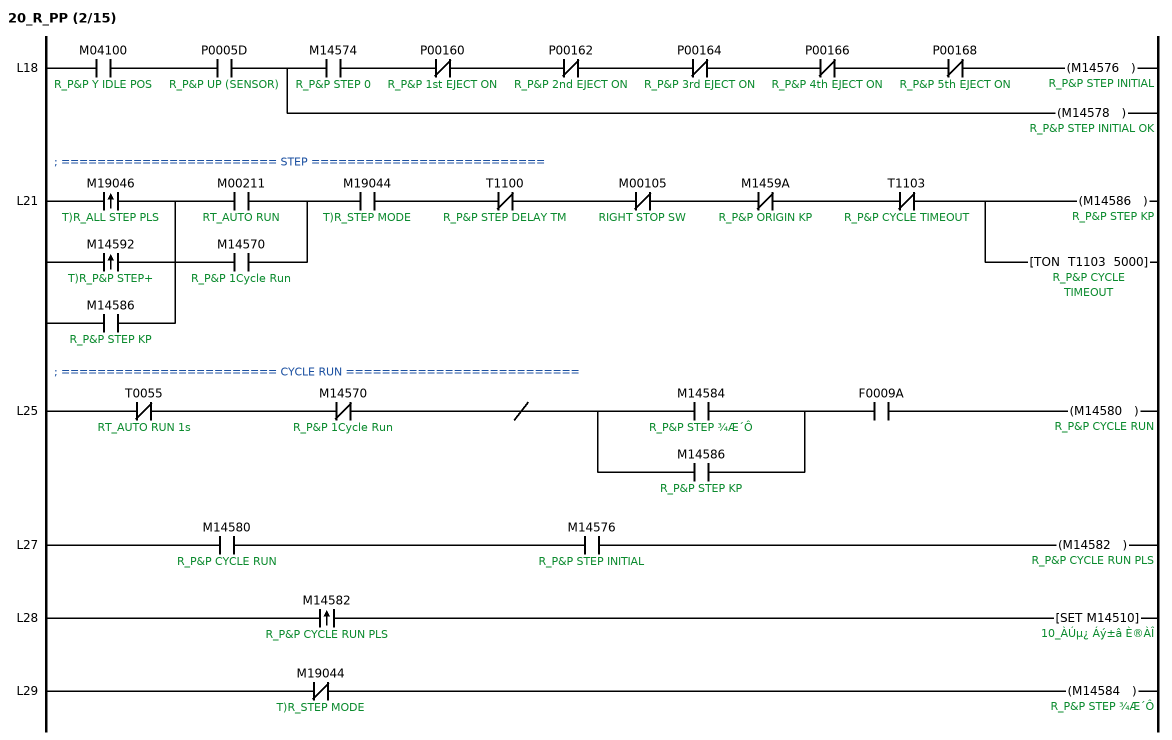
[picture p192: 20_R_PP rungs L18-L29]
; L18
LOAD      M04100	// R_P&P Y IDLE POS
AND       P0005D	// R_P&P UP (SENSOR)
MPUSH
AND       M14574	// R_P&P STEP 0
AND NOT   P00160	// R_P&P 1st EJECT ON
AND NOT   P00162	// R_P&P 2nd EJECT ON
AND NOT   P00164	// R_P&P 3rd EJECT ON
AND NOT   P00166	// R_P&P 4th EJECT ON
AND NOT   P00168	// R_P&P 5th EJECT ON
OUT       M14576	// R_P&P STEP INITIAL
MPOP
OUT       M14578	// R_P&P STEP INITIAL OK
// ======================== STEP ==========================
; L21
LOADP     M19046	// T)R_ALL STEP PLS
ORP       M14592	// T)R_P&P STEP+
OR        M14586	// R_P&P STEP KP
LOAD      M00211	// RT_AUTO RUN
OR        M14570	// R_P&P 1Cycle Run
AND LOAD
AND       M19044	// T)R_STEP MODE
AND NOT   T1100	// R_P&P STEP DELAY TM
AND NOT   M00105	// RIGHT STOP SW
AND NOT   M1459A	// R_P&P ORIGIN KP
AND NOT   T1103	// R_P&P CYCLE TIMEOUT
OUT       M14586	// R_P&P STEP KP
TON       T1103 5000	// R_P&P CYCLE TIMEOUT
// ======================== CYCLE RUN ==========================
; L25
LOAD NOT  T0055	// RT_AUTO RUN 1s
AND NOT   M14570	// R_P&P 1Cycle Run
NOT
LOAD      M14584	// R_P&P STEP ¾Æ´Ô
OR        M14586	// R_P&P STEP KP
AND LOAD
AND       F0009A
OUT       M14580	// R_P&P CYCLE RUN
; L27
LOAD      M14580	// R_P&P CYCLE RUN
AND       M14576	// R_P&P STEP INITIAL
OUT       M14582	// R_P&P CYCLE RUN PLS
; L28
LOADP     M14582	// R_P&P CYCLE RUN PLS
SET       M14510	// 10_ÀÚµ¿ Áý±â È®ÀÎ
; L29
LOAD NOT  M19044	// T)R_STEP MODE
OUT       M14584	// R_P&P STEP ¾Æ´Ô

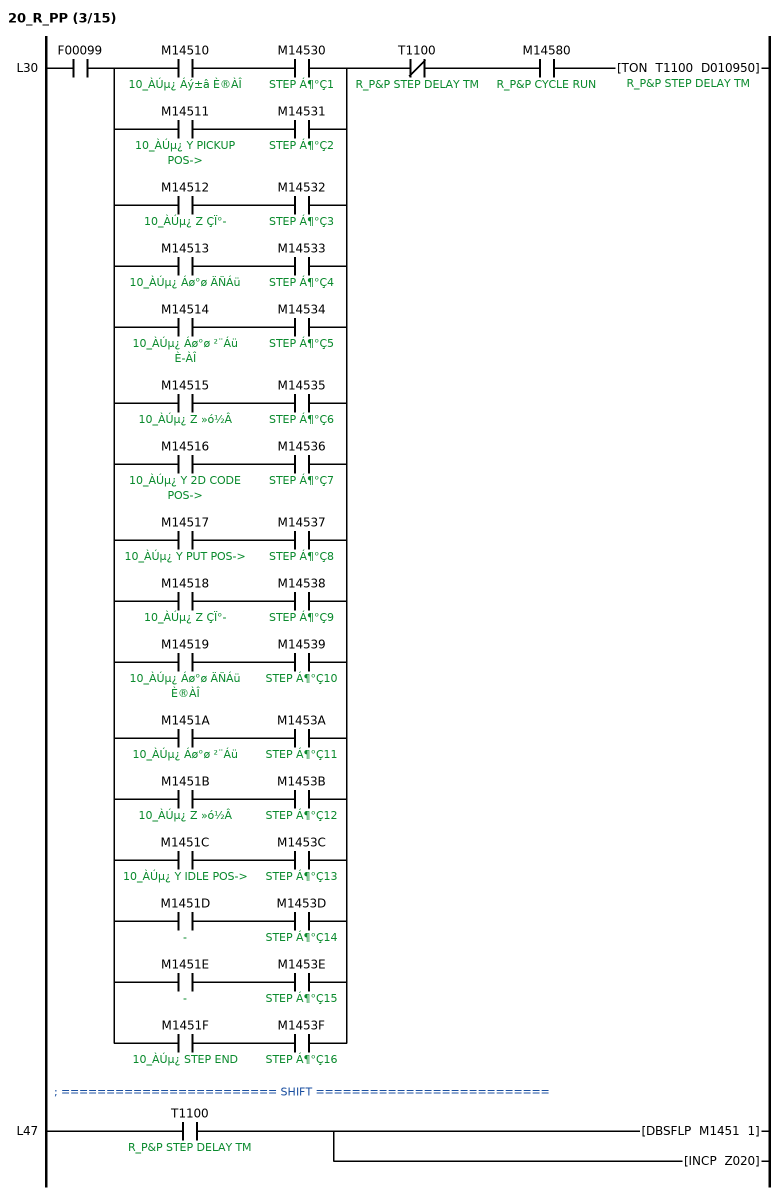
; L30
LOAD      F00099
LOAD      M14510	// 10_ÀÚµ¿ Áý±â È®ÀÎ
AND       M14530	// STEP Á¶°Ç1
LOAD      M14511	// 10_ÀÚµ¿ Y PICKUP POS->
AND       M14531	// STEP Á¶°Ç2
OR LOAD
LOAD      M14512	// 10_ÀÚµ¿ Z ÇÏ°­
AND       M14532	// STEP Á¶°Ç3
OR LOAD
LOAD      M14513	// 10_ÀÚµ¿ Áø°ø ÄÑÁü
AND       M14533	// STEP Á¶°Ç4
OR LOAD
LOAD      M14514	// 10_ÀÚµ¿ Áø°ø ²¨Áü È­ÀÎ
AND       M14534	// STEP Á¶°Ç5
OR LOAD
LOAD      M14515	// 10_ÀÚµ¿ Z »ó½Â
AND       M14535	// STEP Á¶°Ç6
OR LOAD
LOAD      M14516	// 10_ÀÚµ¿ Y 2D CODE POS->
AND       M14536	// STEP Á¶°Ç7
OR LOAD
LOAD      M14517	// 10_ÀÚµ¿ Y PUT POS->
AND       M14537	// STEP Á¶°Ç8
OR LOAD
LOAD      M14518	// 10_ÀÚµ¿ Z ÇÏ°­
AND       M14538	// STEP Á¶°Ç9
OR LOAD
LOAD      M14519	// 10_ÀÚµ¿ Áø°ø ÄÑÁü È®ÀÎ
AND       M14539	// STEP Á¶°Ç10
OR LOAD
LOAD      M1451A	// 10_ÀÚµ¿ Áø°ø ²¨Áü
AND       M1453A	// STEP Á¶°Ç11
OR LOAD
LOAD      M1451B	// 10_ÀÚµ¿ Z »ó½Â
AND       M1453B	// STEP Á¶°Ç12
OR LOAD
LOAD      M1451C	// 10_ÀÚµ¿ Y IDLE POS->
AND       M1453C	// STEP Á¶°Ç13
OR LOAD
LOAD      M1451D	// -
AND       M1453D	// STEP Á¶°Ç14
OR LOAD
LOAD      M1451E	// -
AND       M1453E	// STEP Á¶°Ç15
OR LOAD
LOAD      M1451F	// 10_ÀÚµ¿ STEP END
AND       M1453F	// STEP Á¶°Ç16
OR LOAD
AND LOAD
AND NOT   T1100	// R_P&P STEP DELAY TM
AND       M14580	// R_P&P CYCLE RUN
TON       T1100 D010950	// R_P&P STEP DELAY TM
// ======================== SHIFT ==========================
; L47
LOAD      T1100	// R_P&P STEP DELAY TM
DBSFLP    M1451 1
INCP      Z020

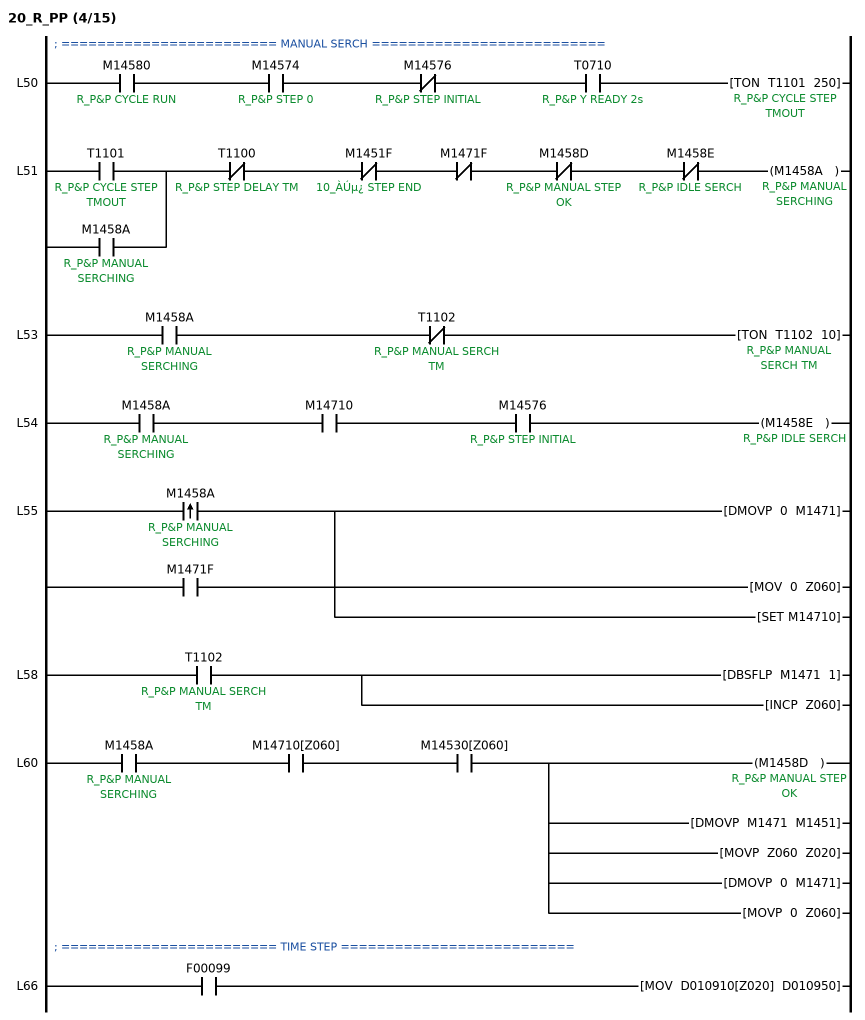
// ======================== MANUAL SERCH ==========================
; L50
LOAD      M14580	// R_P&P CYCLE RUN
AND       M14574	// R_P&P STEP 0
AND NOT   M14576	// R_P&P STEP INITIAL
AND       T0710	// R_P&P Y READY 2s
TON       T1101 250	// R_P&P CYCLE STEP TMOUT
; L51
LOAD      T1101	// R_P&P CYCLE STEP TMOUT
OR        M1458A	// R_P&P MANUAL SERCHING
AND NOT   T1100	// R_P&P STEP DELAY TM
AND NOT   M1451F	// 10_ÀÚµ¿ STEP END
AND NOT   M1471F
AND NOT   M1458D	// R_P&P MANUAL STEP OK
AND NOT   M1458E	// R_P&P IDLE SERCH
OUT       M1458A	// R_P&P MANUAL SERCHING
; L53
LOAD      M1458A	// R_P&P MANUAL SERCHING
AND NOT   T1102	// R_P&P MANUAL SERCH TM
TON       T1102 10	// R_P&P MANUAL SERCH TM
; L54
LOAD      M1458A	// R_P&P MANUAL SERCHING
AND       M14710
AND       M14576	// R_P&P STEP INITIAL
OUT       M1458E	// R_P&P IDLE SERCH
; L55
LOADP     M1458A	// R_P&P MANUAL SERCHING
OR        M1471F
DMOVP     0 M1471
MOV       0 Z060
SET       M14710
; L58
LOAD      T1102	// R_P&P MANUAL SERCH TM
DBSFLP    M1471 1
INCP      Z060
; L60
LOAD      M1458A	// R_P&P MANUAL SERCHING
AND       M14710[Z060]
AND       M14530[Z060]
OUT       M1458D	// R_P&P MANUAL STEP OK
DMOVP     M1471 M1451
MOVP      Z060 Z020
DMOVP     0 M1471
MOVP      0 Z060
// ======================== TIME STEP ==========================
; L66
LOAD      F00099
MOV       D010910[Z020] D010950

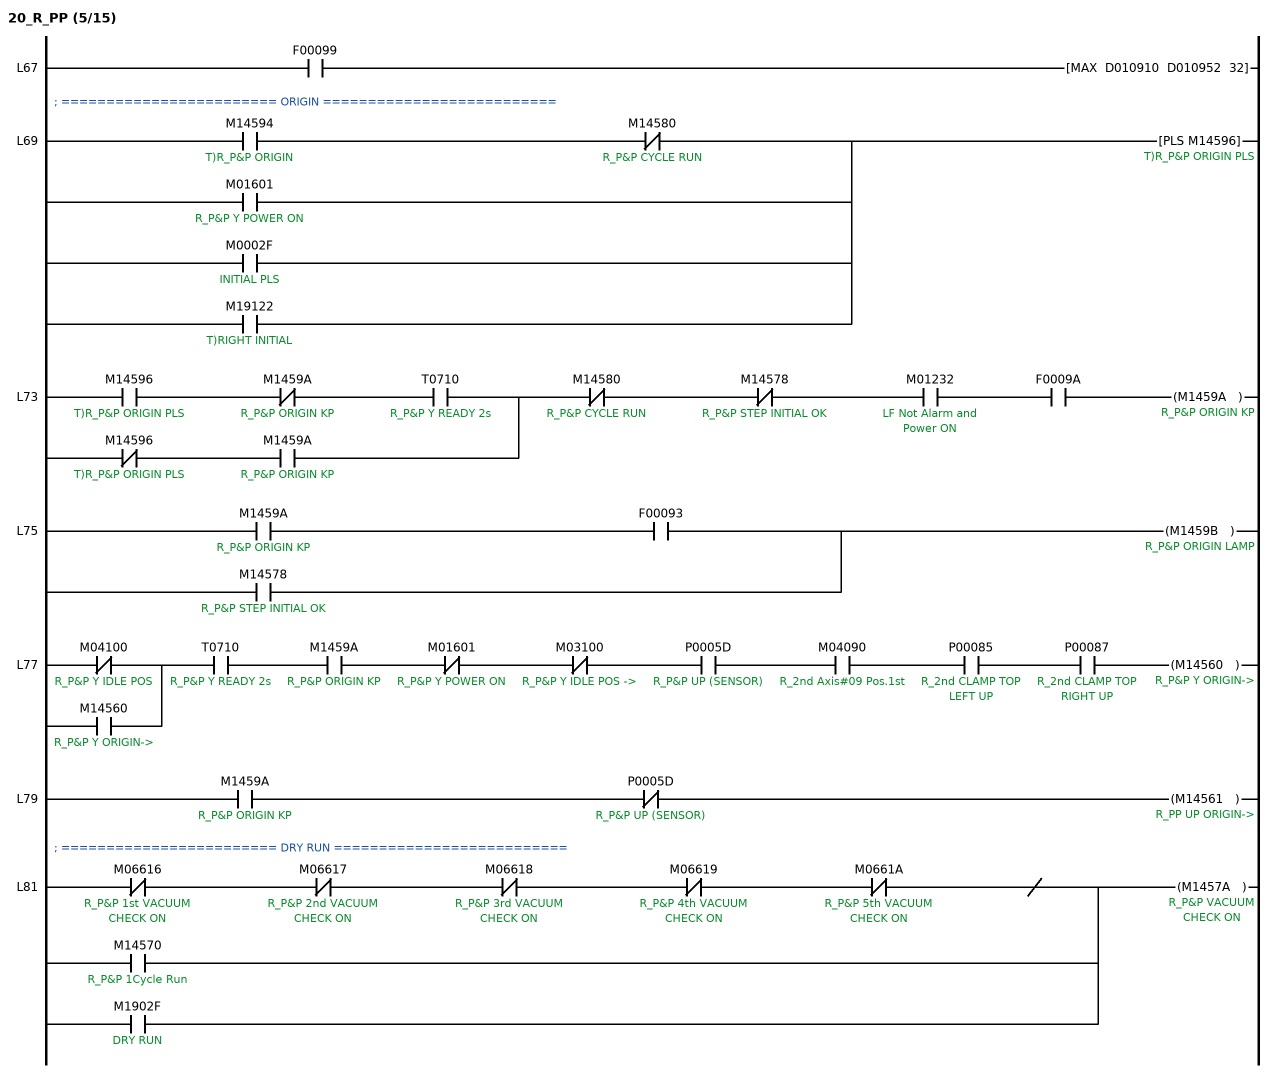
; L67
LOAD      F00099
MAX       D010910 D010952 32
// ======================== ORIGIN ==========================
; L69
LOAD      M14594	// T)R_P&P ORIGIN
AND NOT   M14580	// R_P&P CYCLE RUN
OR        M01601	// R_P&P Y POWER ON
OR        M0002F	// INITIAL PLS
OR        M19122	// T)RIGHT INITIAL
OUTP      M14596	// T)R_P&P ORIGIN PLS
; L73
LOAD      M14596	// T)R_P&P ORIGIN PLS
AND NOT   M1459A	// R_P&P ORIGIN KP
AND       T0710	// R_P&P Y READY 2s
LOAD NOT  M14596	// T)R_P&P ORIGIN PLS
AND       M1459A	// R_P&P ORIGIN KP
OR LOAD
AND NOT   M14580	// R_P&P CYCLE RUN
AND NOT   M14578	// R_P&P STEP INITIAL OK
AND       M01232	// LF Not Alarm and Power ON
AND       F0009A
OUT       M1459A	// R_P&P ORIGIN KP
; L75
LOAD      M1459A	// R_P&P ORIGIN KP
AND       F00093
OR        M14578	// R_P&P STEP INITIAL OK
OUT       M1459B	// R_P&P ORIGIN LAMP
; L77
LOAD NOT  M04100	// R_P&P Y IDLE POS
OR        M14560	// R_P&P Y ORIGIN->
AND       T0710	// R_P&P Y READY 2s
AND       M1459A	// R_P&P ORIGIN KP
AND NOT   M01601	// R_P&P Y POWER ON
AND NOT   M03100	// R_P&P Y IDLE POS ->
AND       P0005D	// R_P&P UP (SENSOR)
AND       M04090	// R_2nd Axis#09 Pos.1st
AND       P00085	// R_2nd CLAMP TOP LEFT UP
AND       P00087	// R_2nd CLAMP TOP RIGHT UP
OUT       M14560	// R_P&P Y ORIGIN->
; L79
LOAD      M1459A	// R_P&P ORIGIN KP
AND NOT   P0005D	// R_P&P UP (SENSOR)
OUT       M14561	// R_PP UP ORIGIN->
// ======================== DRY RUN ==========================
; L81
LOAD NOT  M06616	// R_P&P 1st VACUUM CHECK ON
AND NOT   M06617	// R_P&P 2nd VACUUM CHECK ON
AND NOT   M06618	// R_P&P 3rd VACUUM CHECK ON
AND NOT   M06619	// R_P&P 4th VACUUM CHECK ON
AND NOT   M0661A	// R_P&P 5th VACUUM CHECK ON
NOT
OR        M14570	// R_P&P 1Cycle Run
OR        M1902F	// DRY RUN
OUT       M1457A	// R_P&P VACUUM CHECK ON

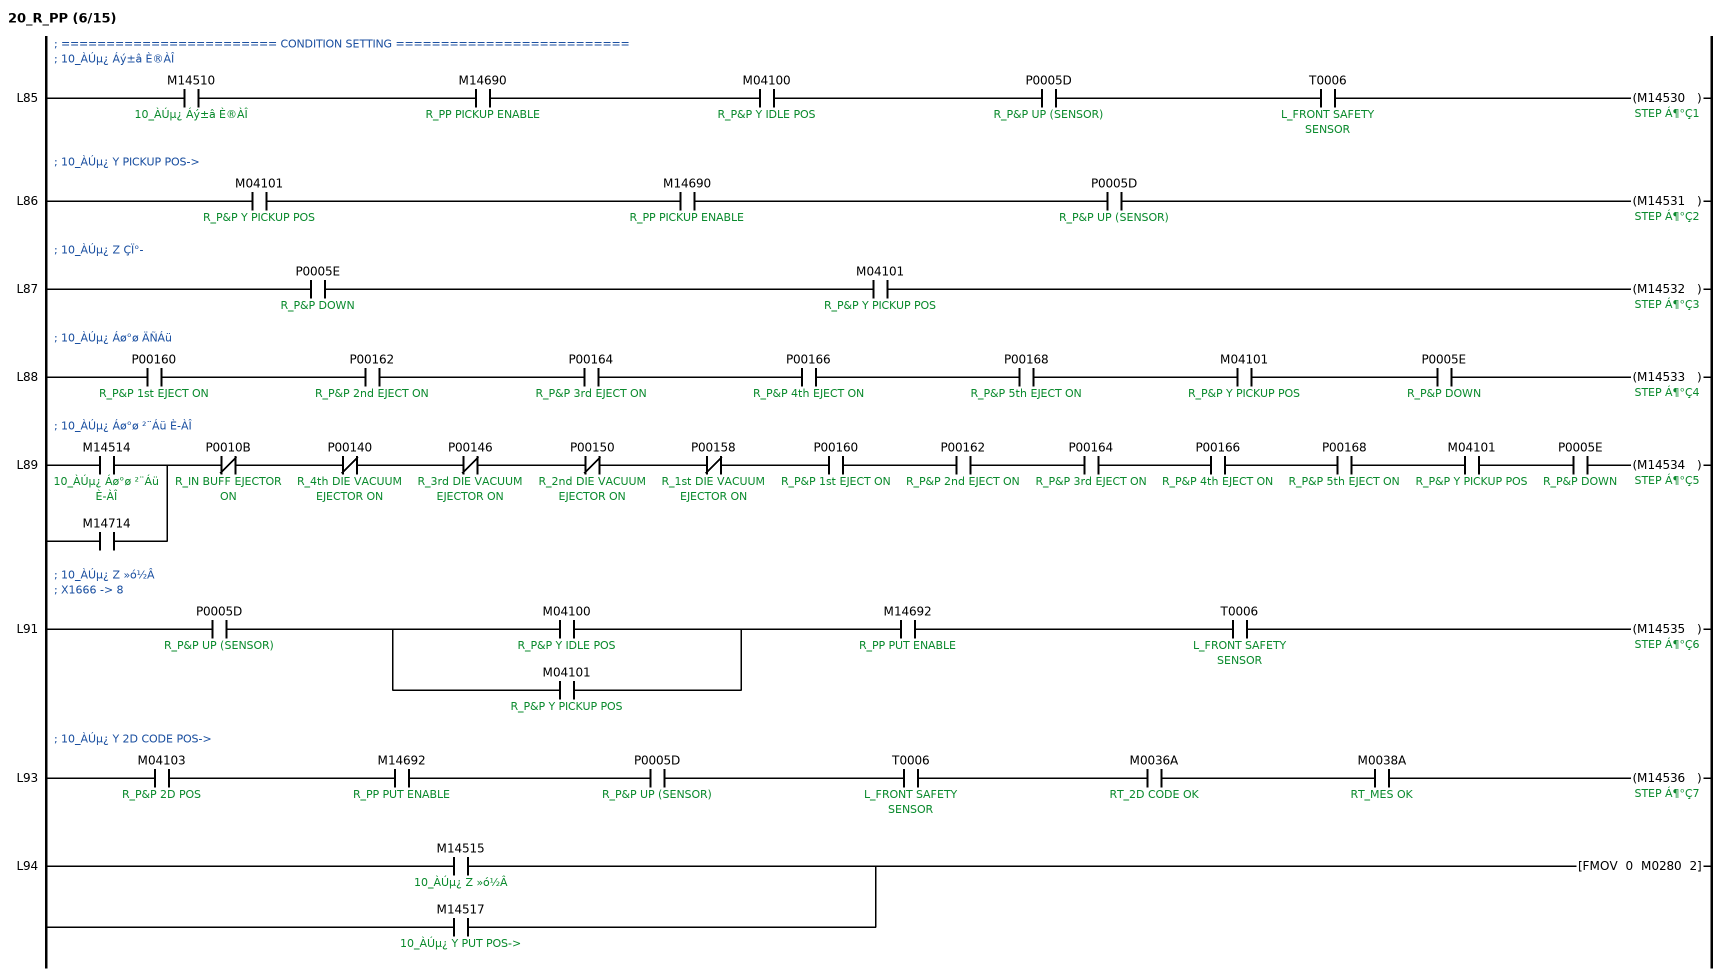
// ======================== CONDITION SETTING ==========================
; L85
LOAD      M14510	// 10_ÀÚµ¿ Áý±â È®ÀÎ
AND       M14690	// R_PP PICKUP ENABLE
AND       M04100	// R_P&P Y IDLE POS
AND       P0005D	// R_P&P UP (SENSOR)
AND       T0006	// L_FRONT SAFETY SENSOR
OUT       M14530	// STEP Á¶°Ç1
// output comment: 10_ÀÚµ¿ Áý±â È®ÀÎ
; L86
LOAD      M04101	// R_P&P Y PICKUP POS
AND       M14690	// R_PP PICKUP ENABLE
AND       P0005D	// R_P&P UP (SENSOR)
OUT       M14531	// STEP Á¶°Ç2
// output comment: 10_ÀÚµ¿ Y PICKUP POS->
; L87
LOAD      P0005E	// R_P&P DOWN
AND       M04101	// R_P&P Y PICKUP POS
OUT       M14532	// STEP Á¶°Ç3
// output comment: 10_ÀÚµ¿ Z ÇÏ°­
; L88
LOAD      P00160	// R_P&P 1st EJECT ON
AND       P00162	// R_P&P 2nd EJECT ON
AND       P00164	// R_P&P 3rd EJECT ON
AND       P00166	// R_P&P 4th EJECT ON
AND       P00168	// R_P&P 5th EJECT ON
AND       M04101	// R_P&P Y PICKUP POS
AND       P0005E	// R_P&P DOWN
OUT       M14533	// STEP Á¶°Ç4
// output comment: 10_ÀÚµ¿ Áø°ø ÄÑÁü
; L89
LOAD      M14514	// 10_ÀÚµ¿ Áø°ø ²¨Áü È­ÀÎ
OR        M14714
AND NOT   P0010B	// R_IN BUFF EJECTOR ON
AND NOT   P00140	// R_4th DIE VACUUM EJECTOR ON
AND NOT   P00146	// R_3rd DIE VACUUM EJECTOR ON
AND NOT   P00150	// R_2nd DIE VACUUM EJECTOR ON
AND NOT   P00158	// R_1st DIE VACUUM EJECTOR ON
AND       P00160	// R_P&P 1st EJECT ON
AND       P00162	// R_P&P 2nd EJECT ON
AND       P00164	// R_P&P 3rd EJECT ON
AND       P00166	// R_P&P 4th EJECT ON
AND       P00168	// R_P&P 5th EJECT ON
AND       M04101	// R_P&P Y PICKUP POS
AND       P0005E	// R_P&P DOWN
OUT       M14534	// STEP Á¶°Ç5
// output comment: 10_ÀÚµ¿ Áø°ø ²¨Áü È­ÀÎ
; L91
LOAD      P0005D	// R_P&P UP (SENSOR)
LOAD      M04100	// R_P&P Y IDLE POS
OR        M04101	// R_P&P Y PICKUP POS
AND LOAD
AND       M14692	// R_PP PUT ENABLE
AND       T0006	// L_FRONT SAFETY SENSOR
OUT       M14535	// STEP Á¶°Ç6
// output comment: 10_ÀÚµ¿ Z »ó½Â X1666 -> 8
; L93
LOAD      M04103	// R_P&P 2D POS
AND       M14692	// R_PP PUT ENABLE
AND       P0005D	// R_P&P UP (SENSOR)
AND       T0006	// L_FRONT SAFETY SENSOR
AND       M0036A	// RT_2D CODE OK
AND       M0038A	// RT_MES OK
OUT       M14536	// STEP Á¶°Ç7
// output comment: 10_ÀÚµ¿ Y 2D CODE POS->
; L94
LOAD      M14515	// 10_ÀÚµ¿ Z »ó½Â
OR        M14517	// 10_ÀÚµ¿ Y PUT POS->
FMOV      0 M0280 2

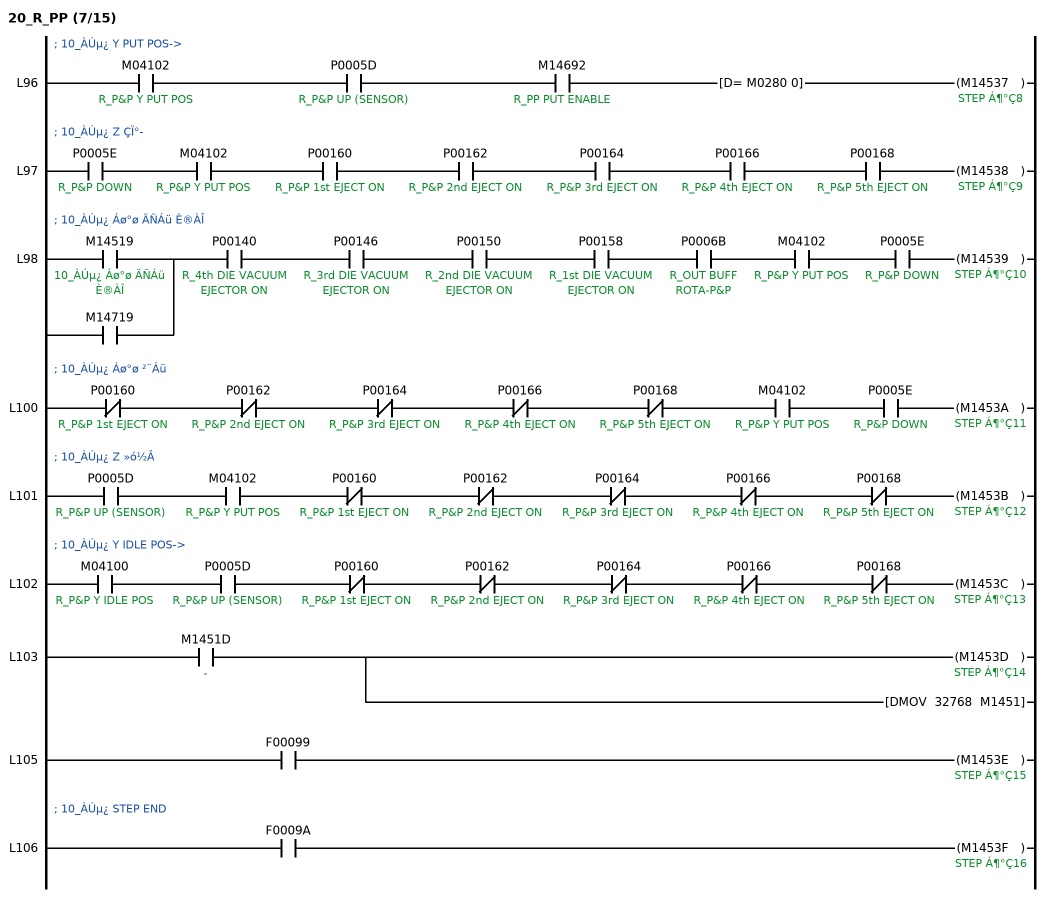
; L96
LOAD      M04102	// R_P&P Y PUT POS
AND       P0005D	// R_P&P UP (SENSOR)
AND       M14692	// R_PP PUT ENABLE
ANDD=     M0280 0
OUT       M14537	// STEP Á¶°Ç8
// output comment: 10_ÀÚµ¿ Y PUT POS->
; L97
LOAD      P0005E	// R_P&P DOWN
AND       M04102	// R_P&P Y PUT POS
AND       P00160	// R_P&P 1st EJECT ON
AND       P00162	// R_P&P 2nd EJECT ON
AND       P00164	// R_P&P 3rd EJECT ON
AND       P00166	// R_P&P 4th EJECT ON
AND       P00168	// R_P&P 5th EJECT ON
OUT       M14538	// STEP Á¶°Ç9
// output comment: 10_ÀÚµ¿ Z ÇÏ°­
; L98
LOAD      M14519	// 10_ÀÚµ¿ Áø°ø ÄÑÁü È®ÀÎ
OR        M14719
AND       P00140	// R_4th DIE VACUUM EJECTOR ON
AND       P00146	// R_3rd DIE VACUUM EJECTOR ON
AND       P00150	// R_2nd DIE VACUUM EJECTOR ON
AND       P00158	// R_1st DIE VACUUM EJECTOR ON
AND       P0006B	// R_OUT BUFF ROTA-P&P
AND       M04102	// R_P&P Y PUT POS
AND       P0005E	// R_P&P DOWN
OUT       M14539	// STEP Á¶°Ç10
// output comment: 10_ÀÚµ¿ Áø°ø ÄÑÁü È®ÀÎ
; L100
LOAD NOT  P00160	// R_P&P 1st EJECT ON
AND NOT   P00162	// R_P&P 2nd EJECT ON
AND NOT   P00164	// R_P&P 3rd EJECT ON
AND NOT   P00166	// R_P&P 4th EJECT ON
AND NOT   P00168	// R_P&P 5th EJECT ON
AND       M04102	// R_P&P Y PUT POS
AND       P0005E	// R_P&P DOWN
OUT       M1453A	// STEP Á¶°Ç11
// output comment: 10_ÀÚµ¿ Áø°ø ²¨Áü
; L101
LOAD      P0005D	// R_P&P UP (SENSOR)
AND       M04102	// R_P&P Y PUT POS
AND NOT   P00160	// R_P&P 1st EJECT ON
AND NOT   P00162	// R_P&P 2nd EJECT ON
AND NOT   P00164	// R_P&P 3rd EJECT ON
AND NOT   P00166	// R_P&P 4th EJECT ON
AND NOT   P00168	// R_P&P 5th EJECT ON
OUT       M1453B	// STEP Á¶°Ç12
// output comment: 10_ÀÚµ¿ Z »ó½Â
; L102
LOAD      M04100	// R_P&P Y IDLE POS
AND       P0005D	// R_P&P UP (SENSOR)
AND NOT   P00160	// R_P&P 1st EJECT ON
AND NOT   P00162	// R_P&P 2nd EJECT ON
AND NOT   P00164	// R_P&P 3rd EJECT ON
AND NOT   P00166	// R_P&P 4th EJECT ON
AND NOT   P00168	// R_P&P 5th EJECT ON
OUT       M1453C	// STEP Á¶°Ç13
// output comment: 10_ÀÚµ¿ Y IDLE POS->
; L103
LOAD      M1451D	// -
OUT       M1453D	// STEP Á¶°Ç14
DMOV      32768 M1451
; L105
LOAD      F00099
OUT       M1453E	// STEP Á¶°Ç15
; L106
LOAD      F0009A
OUT       M1453F	// STEP Á¶°Ç16
// output comment: 10_ÀÚµ¿ STEP END

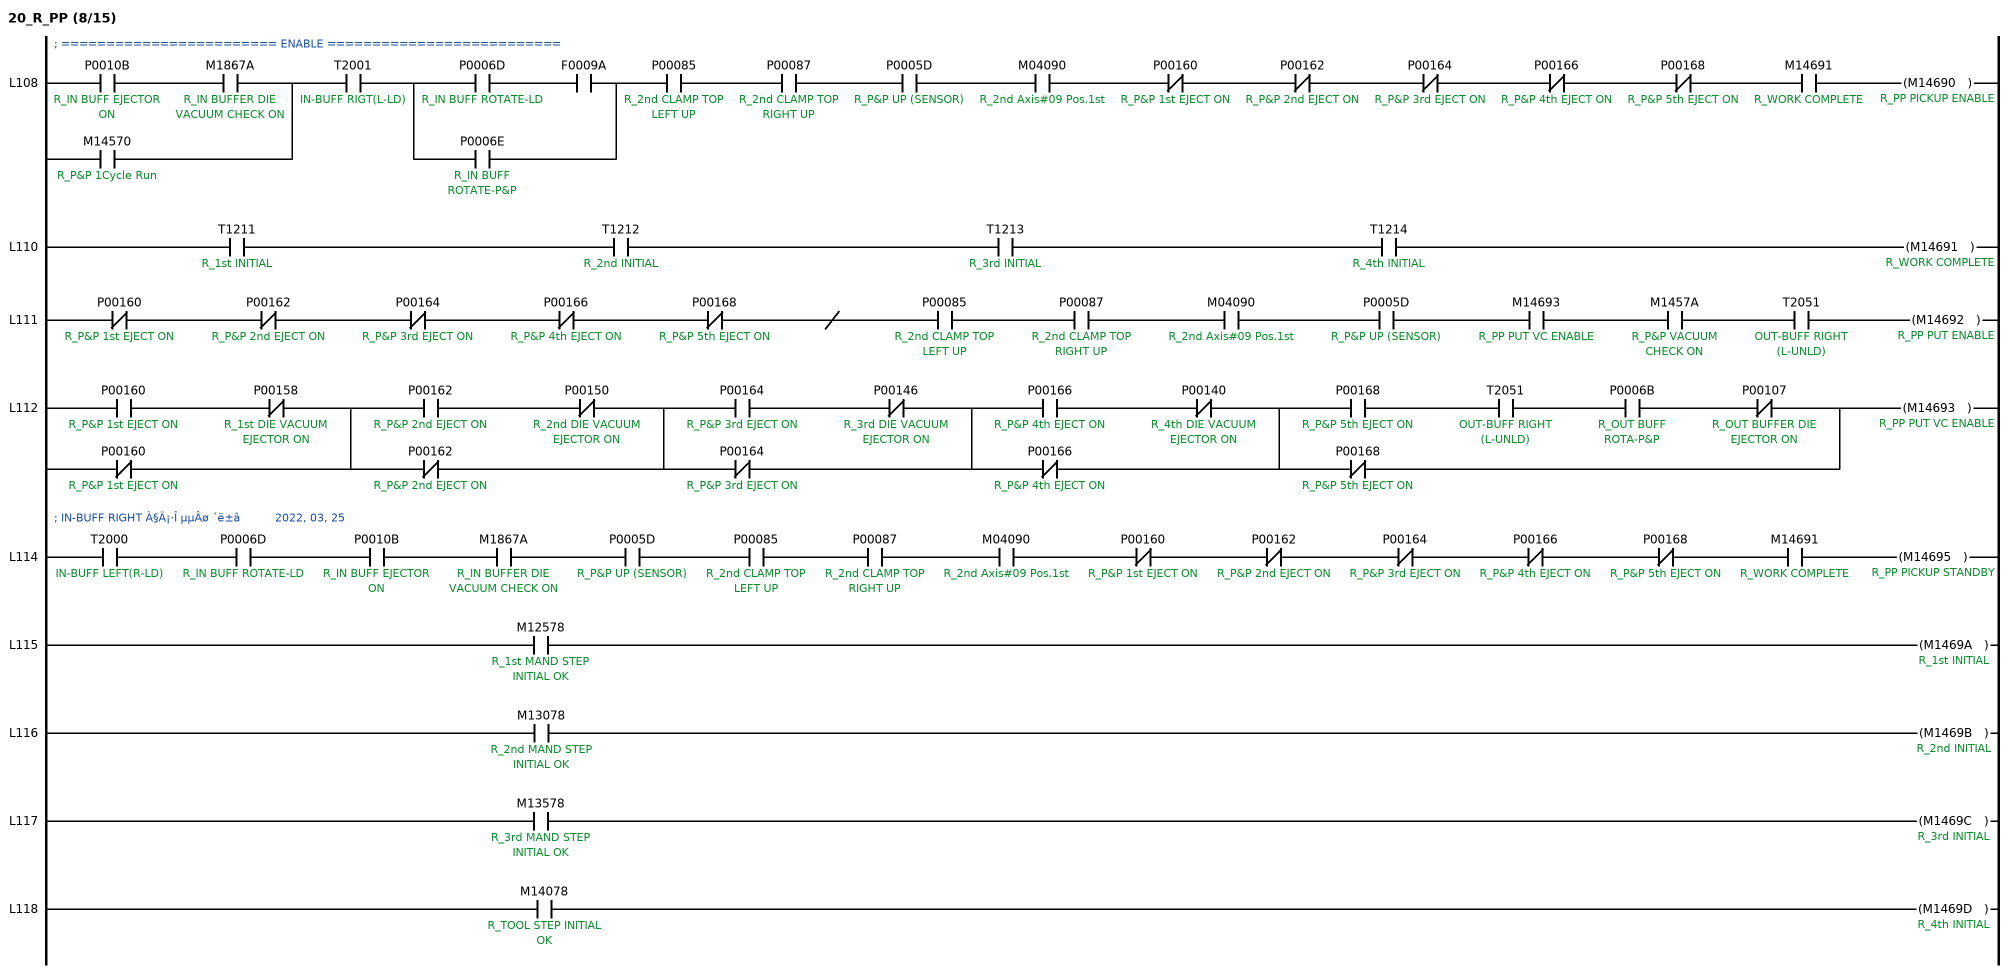
// ======================== ENABLE ==========================
; L108
LOAD      P0010B	// R_IN BUFF EJECTOR ON
AND       M1867A	// R_IN BUFFER DIE VACUUM CHECK ON
OR        M14570	// R_P&P 1Cycle Run
AND       T2001	// IN-BUFF RIGT(L-LD)
LOAD      P0006D	// R_IN BUFF ROTATE-LD
AND       F0009A
OR        P0006E	// R_IN BUFF ROTATE-P&P
AND LOAD
AND       P00085	// R_2nd CLAMP TOP LEFT UP
AND       P00087	// R_2nd CLAMP TOP RIGHT UP
AND       P0005D	// R_P&P UP (SENSOR)
AND       M04090	// R_2nd Axis#09 Pos.1st
AND NOT   P00160	// R_P&P 1st EJECT ON
AND NOT   P00162	// R_P&P 2nd EJECT ON
AND NOT   P00164	// R_P&P 3rd EJECT ON
AND NOT   P00166	// R_P&P 4th EJECT ON
AND NOT   P00168	// R_P&P 5th EJECT ON
AND       M14691	// R_WORK COMPLETE
OUT       M14690	// R_PP PICKUP ENABLE
; L110
LOAD      T1211	// R_1st INITIAL
AND       T1212	// R_2nd INITIAL
AND       T1213	// R_3rd INITIAL
AND       T1214	// R_4th INITIAL
OUT       M14691	// R_WORK COMPLETE
; L111
LOAD NOT  P00160	// R_P&P 1st EJECT ON
AND NOT   P00162	// R_P&P 2nd EJECT ON
AND NOT   P00164	// R_P&P 3rd EJECT ON
AND NOT   P00166	// R_P&P 4th EJECT ON
AND NOT   P00168	// R_P&P 5th EJECT ON
NOT
AND       P00085	// R_2nd CLAMP TOP LEFT UP
AND       P00087	// R_2nd CLAMP TOP RIGHT UP
AND       M04090	// R_2nd Axis#09 Pos.1st
AND       P0005D	// R_P&P UP (SENSOR)
AND       M14693	// R_PP PUT VC ENABLE
AND       M1457A	// R_P&P VACUUM CHECK ON
AND       T2051	// OUT-BUFF RIGHT (L-UNLD)
OUT       M14692	// R_PP PUT ENABLE
; L112
LOAD      P00160	// R_P&P 1st EJECT ON
AND NOT   P00158	// R_1st DIE VACUUM EJECTOR ON
OR NOT    P00160	// R_P&P 1st EJECT ON
LOAD      P00162	// R_P&P 2nd EJECT ON
AND NOT   P00150	// R_2nd DIE VACUUM EJECTOR ON
OR NOT    P00162	// R_P&P 2nd EJECT ON
AND LOAD
LOAD      P00164	// R_P&P 3rd EJECT ON
AND NOT   P00146	// R_3rd DIE VACUUM EJECTOR ON
OR NOT    P00164	// R_P&P 3rd EJECT ON
AND LOAD
LOAD      P00166	// R_P&P 4th EJECT ON
AND NOT   P00140	// R_4th DIE VACUUM EJECTOR ON
OR NOT    P00166	// R_P&P 4th EJECT ON
AND LOAD
LOAD      P00168	// R_P&P 5th EJECT ON
AND       T2051	// OUT-BUFF RIGHT (L-UNLD)
AND       P0006B	// R_OUT BUFF ROTA-P&P
AND NOT   P00107	// R_OUT BUFFER DIE EJECTOR ON
OR NOT    P00168	// R_P&P 5th EJECT ON
AND LOAD
OUT       M14693	// R_PP PUT VC ENABLE
; L114
LOAD      T2000	// IN-BUFF LEFT(R-LD)
AND       P0006D	// R_IN BUFF ROTATE-LD
AND       P0010B	// R_IN BUFF EJECTOR ON
AND       M1867A	// R_IN BUFFER DIE VACUUM CHECK ON
AND       P0005D	// R_P&P UP (SENSOR)
AND       P00085	// R_2nd CLAMP TOP LEFT UP
AND       P00087	// R_2nd CLAMP TOP RIGHT UP
AND       M04090	// R_2nd Axis#09 Pos.1st
AND NOT   P00160	// R_P&P 1st EJECT ON
AND NOT   P00162	// R_P&P 2nd EJECT ON
AND NOT   P00164	// R_P&P 3rd EJECT ON
AND NOT   P00166	// R_P&P 4th EJECT ON
AND NOT   P00168	// R_P&P 5th EJECT ON
AND       M14691	// R_WORK COMPLETE
OUT       M14695	// R_PP PICKUP STANDBY
// output comment: IN-BUFF RIGHT À§Ä¡·Î µµÂø ´ë±â          2022, 03, 25
; L115
LOAD      M12578	// R_1st MAND STEP INITIAL OK
OUT       M1469A	// R_1st INITIAL
; L116
LOAD      M13078	// R_2nd MAND STEP INITIAL OK
OUT       M1469B	// R_2nd INITIAL
; L117
LOAD      M13578	// R_3rd MAND STEP INITIAL OK
OUT       M1469C	// R_3rd INITIAL
; L118
LOAD      M14078	// R_TOOL STEP INITIAL OK
OUT       M1469D	// R_4th INITIAL

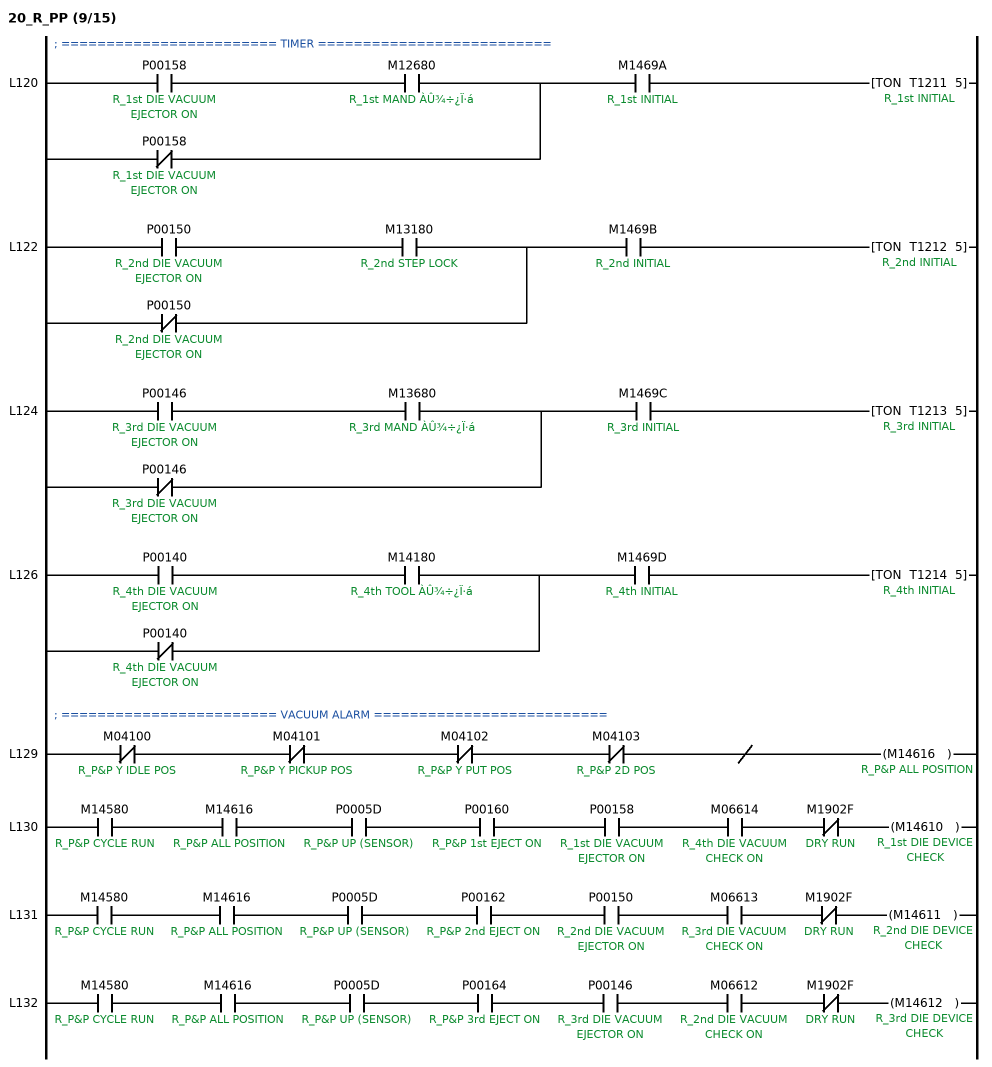
// ======================== TIMER ==========================
; L120
LOAD      P00158	// R_1st DIE VACUUM EJECTOR ON
AND       M12680	// R_1st MAND ÀÛ¾÷¿Ï·á
OR NOT    P00158	// R_1st DIE VACUUM EJECTOR ON
AND       M1469A	// R_1st INITIAL
TON       T1211 5	// R_1st INITIAL
; L122
LOAD      P00150	// R_2nd DIE VACUUM EJECTOR ON
AND       M13180	// R_2nd STEP LOCK
OR NOT    P00150	// R_2nd DIE VACUUM EJECTOR ON
AND       M1469B	// R_2nd INITIAL
TON       T1212 5	// R_2nd INITIAL
; L124
LOAD      P00146	// R_3rd DIE VACUUM EJECTOR ON
AND       M13680	// R_3rd MAND ÀÛ¾÷¿Ï·á
OR NOT    P00146	// R_3rd DIE VACUUM EJECTOR ON
AND       M1469C	// R_3rd INITIAL
TON       T1213 5	// R_3rd INITIAL
; L126
LOAD      P00140	// R_4th DIE VACUUM EJECTOR ON
AND       M14180	// R_4th TOOL ÀÛ¾÷¿Ï·á
OR NOT    P00140	// R_4th DIE VACUUM EJECTOR ON
AND       M1469D	// R_4th INITIAL
TON       T1214 5	// R_4th INITIAL
// ======================== VACUUM ALARM ==========================
; L129
LOAD NOT  M04100	// R_P&P Y IDLE POS
AND NOT   M04101	// R_P&P Y PICKUP POS
AND NOT   M04102	// R_P&P Y PUT POS
AND NOT   M04103	// R_P&P 2D POS
NOT
OUT       M14616	// R_P&P ALL POSITION
; L130
LOAD      M14580	// R_P&P CYCLE RUN
AND       M14616	// R_P&P ALL POSITION
AND       P0005D	// R_P&P UP (SENSOR)
AND       P00160	// R_P&P 1st EJECT ON
AND       P00158	// R_1st DIE VACUUM EJECTOR ON
AND       M06614	// R_4th DIE VACUUM CHECK ON
AND NOT   M1902F	// DRY RUN
OUT       M14610	// R_1st DIE DEVICE CHECK
; L131
LOAD      M14580	// R_P&P CYCLE RUN
AND       M14616	// R_P&P ALL POSITION
AND       P0005D	// R_P&P UP (SENSOR)
AND       P00162	// R_P&P 2nd EJECT ON
AND       P00150	// R_2nd DIE VACUUM EJECTOR ON
AND       M06613	// R_3rd DIE VACUUM CHECK ON
AND NOT   M1902F	// DRY RUN
OUT       M14611	// R_2nd DIE DEVICE CHECK
; L132
LOAD      M14580	// R_P&P CYCLE RUN
AND       M14616	// R_P&P ALL POSITION
AND       P0005D	// R_P&P UP (SENSOR)
AND       P00164	// R_P&P 3rd EJECT ON
AND       P00146	// R_3rd DIE VACUUM EJECTOR ON
AND       M06612	// R_2nd DIE VACUUM CHECK ON
AND NOT   M1902F	// DRY RUN
OUT       M14612	// R_3rd DIE DEVICE CHECK

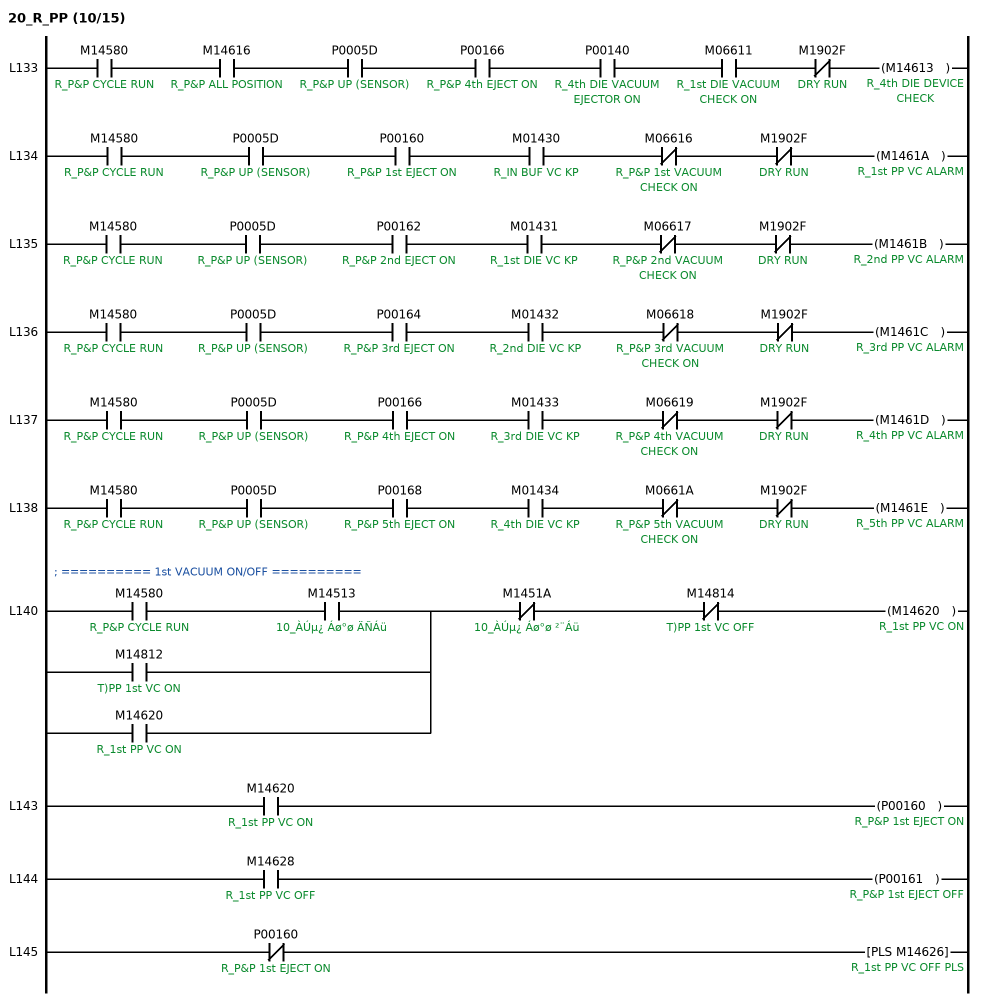
; L133
LOAD      M14580	// R_P&P CYCLE RUN
AND       M14616	// R_P&P ALL POSITION
AND       P0005D	// R_P&P UP (SENSOR)
AND       P00166	// R_P&P 4th EJECT ON
AND       P00140	// R_4th DIE VACUUM EJECTOR ON
AND       M06611	// R_1st DIE VACUUM CHECK ON
AND NOT   M1902F	// DRY RUN
OUT       M14613	// R_4th DIE DEVICE CHECK
; L134
LOAD      M14580	// R_P&P CYCLE RUN
AND       P0005D	// R_P&P UP (SENSOR)
AND       P00160	// R_P&P 1st EJECT ON
AND       M01430	// R_IN BUF VC KP
AND NOT   M06616	// R_P&P 1st VACUUM CHECK ON
AND NOT   M1902F	// DRY RUN
OUT       M1461A	// R_1st PP VC ALARM
; L135
LOAD      M14580	// R_P&P CYCLE RUN
AND       P0005D	// R_P&P UP (SENSOR)
AND       P00162	// R_P&P 2nd EJECT ON
AND       M01431	// R_1st DIE VC KP
AND NOT   M06617	// R_P&P 2nd VACUUM CHECK ON
AND NOT   M1902F	// DRY RUN
OUT       M1461B	// R_2nd PP VC ALARM
; L136
LOAD      M14580	// R_P&P CYCLE RUN
AND       P0005D	// R_P&P UP (SENSOR)
AND       P00164	// R_P&P 3rd EJECT ON
AND       M01432	// R_2nd DIE VC KP
AND NOT   M06618	// R_P&P 3rd VACUUM CHECK ON
AND NOT   M1902F	// DRY RUN
OUT       M1461C	// R_3rd PP VC ALARM
; L137
LOAD      M14580	// R_P&P CYCLE RUN
AND       P0005D	// R_P&P UP (SENSOR)
AND       P00166	// R_P&P 4th EJECT ON
AND       M01433	// R_3rd DIE VC KP
AND NOT   M06619	// R_P&P 4th VACUUM CHECK ON
AND NOT   M1902F	// DRY RUN
OUT       M1461D	// R_4th PP VC ALARM
; L138
LOAD      M14580	// R_P&P CYCLE RUN
AND       P0005D	// R_P&P UP (SENSOR)
AND       P00168	// R_P&P 5th EJECT ON
AND       M01434	// R_4th DIE VC KP
AND NOT   M0661A	// R_P&P 5th VACUUM CHECK ON
AND NOT   M1902F	// DRY RUN
OUT       M1461E	// R_5th PP VC ALARM
// ========== 1st VACUUM ON/OFF ==========
; L140
LOAD      M14580	// R_P&P CYCLE RUN
AND       M14513	// 10_ÀÚµ¿ Áø°ø ÄÑÁü
OR        M14812	// T)PP 1st VC ON
OR        M14620	// R_1st PP VC ON
AND NOT   M1451A	// 10_ÀÚµ¿ Áø°ø ²¨Áü
AND NOT   M14814	// T)PP 1st VC OFF
OUT       M14620	// R_1st PP VC ON
; L143
LOAD      M14620	// R_1st PP VC ON
OUT       P00160	// R_P&P 1st EJECT ON
; L144
LOAD      M14628	// R_1st PP VC OFF
OUT       P00161	// R_P&P 1st EJECT OFF
; L145
LOAD NOT  P00160	// R_P&P 1st EJECT ON
OUTP      M14626	// R_1st PP VC OFF PLS

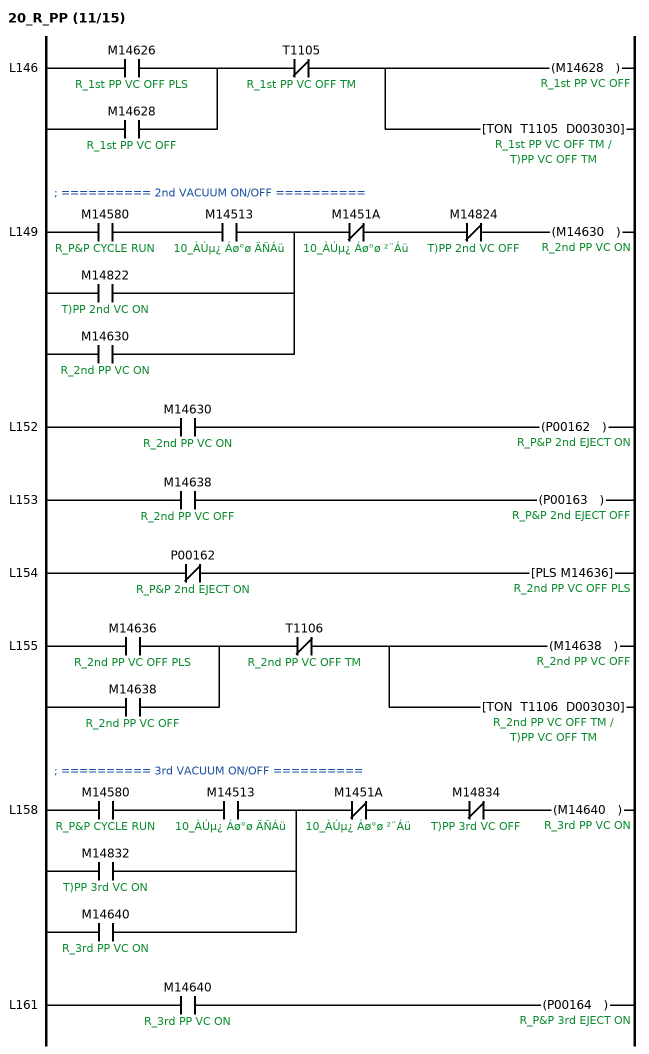
; L146
LOAD      M14626	// R_1st PP VC OFF PLS
OR        M14628	// R_1st PP VC OFF
AND NOT   T1105	// R_1st PP VC OFF TM
OUT       M14628	// R_1st PP VC OFF
TON       T1105 D003030	// R_1st PP VC OFF TM / T)PP VC OFF TM
// ========== 2nd VACUUM ON/OFF ==========
; L149
LOAD      M14580	// R_P&P CYCLE RUN
AND       M14513	// 10_ÀÚµ¿ Áø°ø ÄÑÁü
OR        M14822	// T)PP 2nd VC ON
OR        M14630	// R_2nd PP VC ON
AND NOT   M1451A	// 10_ÀÚµ¿ Áø°ø ²¨Áü
AND NOT   M14824	// T)PP 2nd VC OFF
OUT       M14630	// R_2nd PP VC ON
; L152
LOAD      M14630	// R_2nd PP VC ON
OUT       P00162	// R_P&P 2nd EJECT ON
; L153
LOAD      M14638	// R_2nd PP VC OFF
OUT       P00163	// R_P&P 2nd EJECT OFF
; L154
LOAD NOT  P00162	// R_P&P 2nd EJECT ON
OUTP      M14636	// R_2nd PP VC OFF PLS
; L155
LOAD      M14636	// R_2nd PP VC OFF PLS
OR        M14638	// R_2nd PP VC OFF
AND NOT   T1106	// R_2nd PP VC OFF TM
OUT       M14638	// R_2nd PP VC OFF
TON       T1106 D003030	// R_2nd PP VC OFF TM / T)PP VC OFF TM
// ========== 3rd VACUUM ON/OFF ==========
; L158
LOAD      M14580	// R_P&P CYCLE RUN
AND       M14513	// 10_ÀÚµ¿ Áø°ø ÄÑÁü
OR        M14832	// T)PP 3rd VC ON
OR        M14640	// R_3rd PP VC ON
AND NOT   M1451A	// 10_ÀÚµ¿ Áø°ø ²¨Áü
AND NOT   M14834	// T)PP 3rd VC OFF
OUT       M14640	// R_3rd PP VC ON
; L161
LOAD      M14640	// R_3rd PP VC ON
OUT       P00164	// R_P&P 3rd EJECT ON

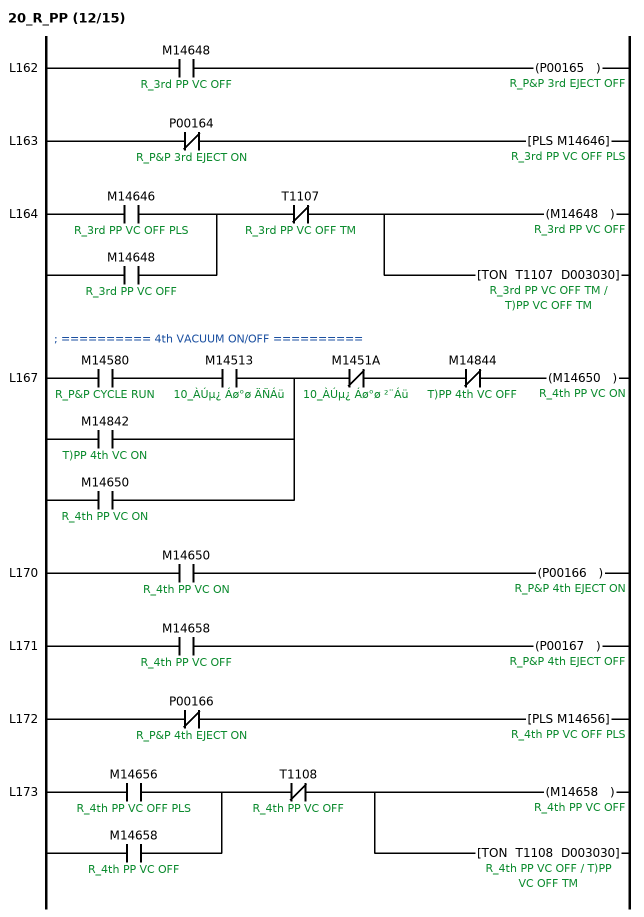
; L162
LOAD      M14648	// R_3rd PP VC OFF
OUT       P00165	// R_P&P 3rd EJECT OFF
; L163
LOAD NOT  P00164	// R_P&P 3rd EJECT ON
OUTP      M14646	// R_3rd PP VC OFF PLS
; L164
LOAD      M14646	// R_3rd PP VC OFF PLS
OR        M14648	// R_3rd PP VC OFF
AND NOT   T1107	// R_3rd PP VC OFF TM
OUT       M14648	// R_3rd PP VC OFF
TON       T1107 D003030	// R_3rd PP VC OFF TM / T)PP VC OFF TM
// ========== 4th VACUUM ON/OFF ==========
; L167
LOAD      M14580	// R_P&P CYCLE RUN
AND       M14513	// 10_ÀÚµ¿ Áø°ø ÄÑÁü
OR        M14842	// T)PP 4th VC ON
OR        M14650	// R_4th PP VC ON
AND NOT   M1451A	// 10_ÀÚµ¿ Áø°ø ²¨Áü
AND NOT   M14844	// T)PP 4th VC OFF
OUT       M14650	// R_4th PP VC ON
; L170
LOAD      M14650	// R_4th PP VC ON
OUT       P00166	// R_P&P 4th EJECT ON
; L171
LOAD      M14658	// R_4th PP VC OFF
OUT       P00167	// R_P&P 4th EJECT OFF
; L172
LOAD NOT  P00166	// R_P&P 4th EJECT ON
OUTP      M14656	// R_4th PP VC OFF PLS
; L173
LOAD      M14656	// R_4th PP VC OFF PLS
OR        M14658	// R_4th PP VC OFF
AND NOT   T1108	// R_4th PP VC OFF
OUT       M14658	// R_4th PP VC OFF
TON       T1108 D003030	// R_4th PP VC OFF / T)PP VC OFF TM

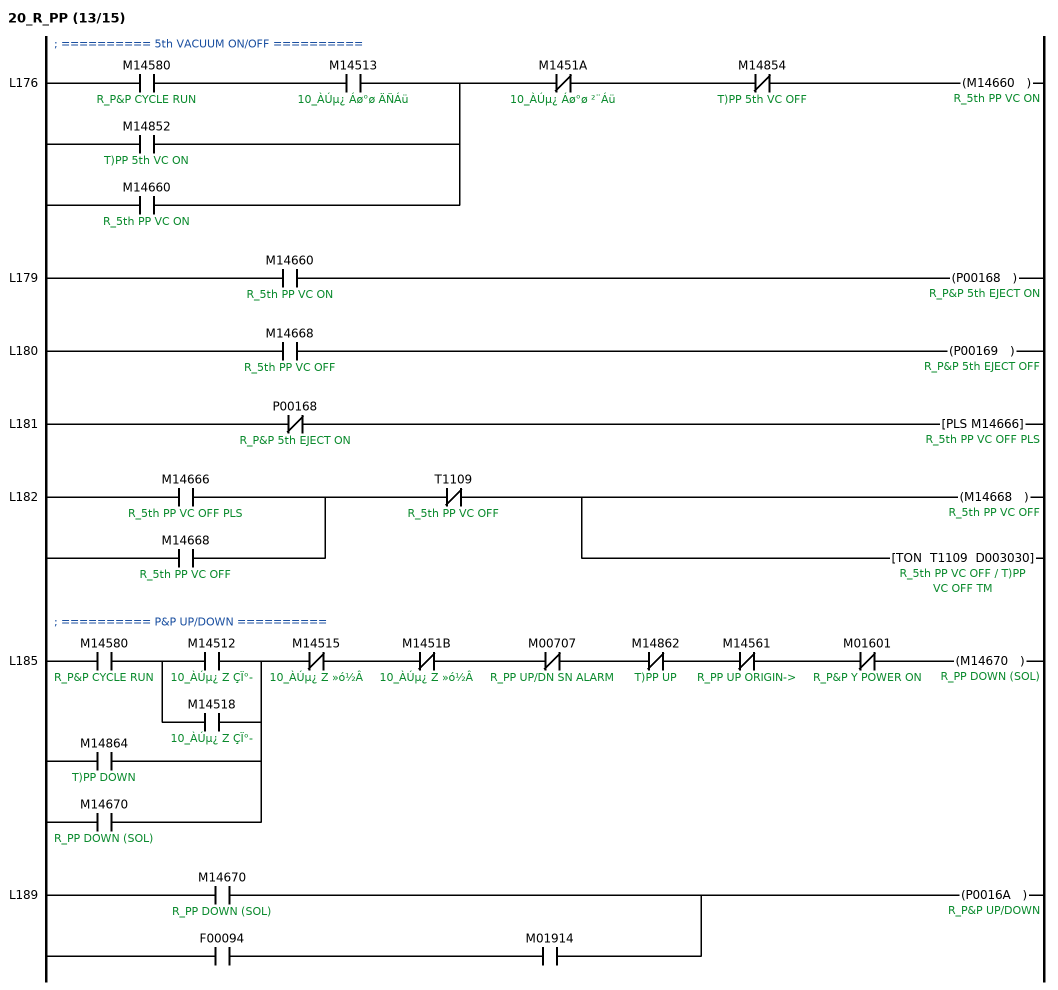
// ========== 5th VACUUM ON/OFF ==========
; L176
LOAD      M14580	// R_P&P CYCLE RUN
AND       M14513	// 10_ÀÚµ¿ Áø°ø ÄÑÁü
OR        M14852	// T)PP 5th VC ON
OR        M14660	// R_5th PP VC ON
AND NOT   M1451A	// 10_ÀÚµ¿ Áø°ø ²¨Áü
AND NOT   M14854	// T)PP 5th VC OFF
OUT       M14660	// R_5th PP VC ON
; L179
LOAD      M14660	// R_5th PP VC ON
OUT       P00168	// R_P&P 5th EJECT ON
; L180
LOAD      M14668	// R_5th PP VC OFF
OUT       P00169	// R_P&P 5th EJECT OFF
; L181
LOAD NOT  P00168	// R_P&P 5th EJECT ON
OUTP      M14666	// R_5th PP VC OFF PLS
; L182
LOAD      M14666	// R_5th PP VC OFF PLS
OR        M14668	// R_5th PP VC OFF
AND NOT   T1109	// R_5th PP VC OFF
OUT       M14668	// R_5th PP VC OFF
TON       T1109 D003030	// R_5th PP VC OFF / T)PP VC OFF TM
// ========== P&P UP/DOWN ==========
; L185
LOAD      M14580	// R_P&P CYCLE RUN
LOAD      M14512	// 10_ÀÚµ¿ Z ÇÏ°­
OR        M14518	// 10_ÀÚµ¿ Z ÇÏ°­
AND LOAD
OR        M14864	// T)PP DOWN
OR        M14670	// R_PP DOWN (SOL)
AND NOT   M14515	// 10_ÀÚµ¿ Z »ó½Â
AND NOT   M1451B	// 10_ÀÚµ¿ Z »ó½Â
AND NOT   M00707	// R_PP UP/DN SN ALARM
AND NOT   M14862	// T)PP UP
AND NOT   M14561	// R_PP UP ORIGIN->
AND NOT   M01601	// R_P&P Y POWER ON
OUT       M14670	// R_PP DOWN (SOL)
; L189
LOAD      M14670	// R_PP DOWN (SOL)
LOAD      F00094
AND       M01914
OR LOAD
OUT       P0016A	// R_P&P UP/DOWN

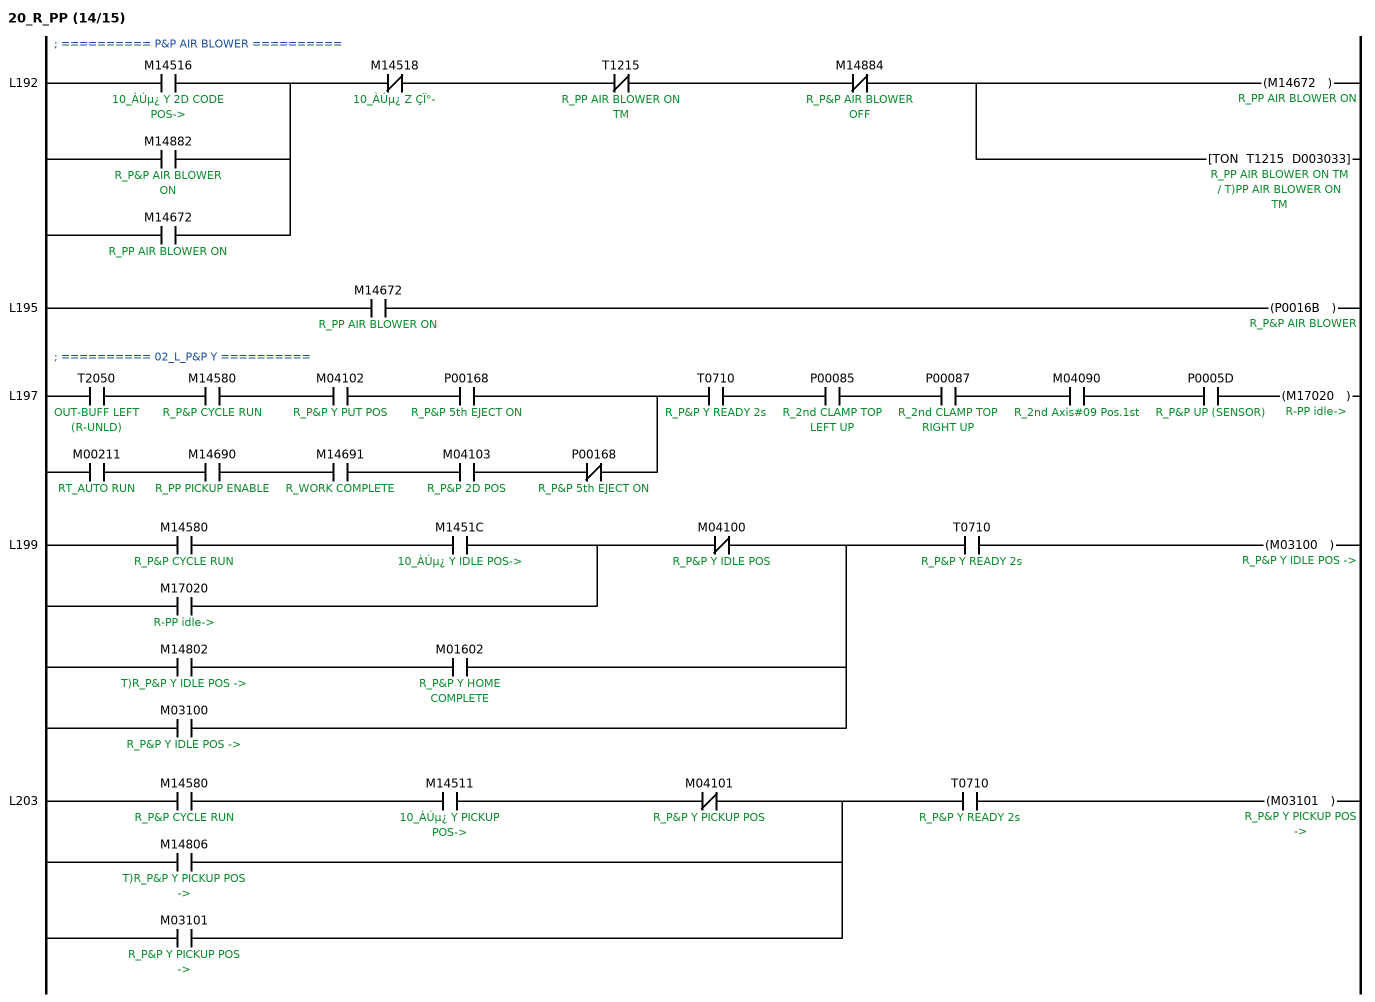
// ========== P&P AIR BLOWER ==========
; L192
LOAD      M14516	// 10_ÀÚµ¿ Y 2D CODE POS->
OR        M14882	// R_P&P AIR BLOWER ON
OR        M14672	// R_PP AIR BLOWER ON
AND NOT   M14518	// 10_ÀÚµ¿ Z ÇÏ°­
AND NOT   T1215	// R_PP AIR BLOWER ON TM
AND NOT   M14884	// R_P&P AIR BLOWER OFF
OUT       M14672	// R_PP AIR BLOWER ON
TON       T1215 D003033	// R_PP AIR BLOWER ON TM / T)PP AIR BLOWER ON TM
; L195
LOAD      M14672	// R_PP AIR BLOWER ON
OUT       P0016B	// R_P&P AIR BLOWER
// ========== 02_L_P&P Y ==========
; L197
LOAD      T2050	// OUT-BUFF LEFT (R-UNLD)
AND       M14580	// R_P&P CYCLE RUN
AND       M04102	// R_P&P Y PUT POS
AND       P00168	// R_P&P 5th EJECT ON
LOAD      M00211	// RT_AUTO RUN
AND       M14690	// R_PP PICKUP ENABLE
AND       M14691	// R_WORK COMPLETE
AND       M04103	// R_P&P 2D POS
AND NOT   P00168	// R_P&P 5th EJECT ON
OR LOAD
AND       T0710	// R_P&P Y READY 2s
AND       P00085	// R_2nd CLAMP TOP LEFT UP
AND       P00087	// R_2nd CLAMP TOP RIGHT UP
AND       M04090	// R_2nd Axis#09 Pos.1st
AND       P0005D	// R_P&P UP (SENSOR)
OUT       M17020	// R-PP idle->
; L199
LOAD      M14580	// R_P&P CYCLE RUN
AND       M1451C	// 10_ÀÚµ¿ Y IDLE POS->
OR        M17020	// R-PP idle->
AND NOT   M04100	// R_P&P Y IDLE POS
LOAD      M14802	// T)R_P&P Y IDLE POS ->
AND       M01602	// R_P&P Y HOME COMPLETE
OR LOAD
OR        M03100	// R_P&P Y IDLE POS ->
AND       T0710	// R_P&P Y READY 2s
OUT       M03100	// R_P&P Y IDLE POS ->
; L203
LOAD      M14580	// R_P&P CYCLE RUN
AND       M14511	// 10_ÀÚµ¿ Y PICKUP POS->
AND NOT   M04101	// R_P&P Y PICKUP POS
OR        M14806	// T)R_P&P Y PICKUP POS ->
OR        M03101	// R_P&P Y PICKUP POS ->
AND       T0710	// R_P&P Y READY 2s
OUT       M03101	// R_P&P Y PICKUP POS ->

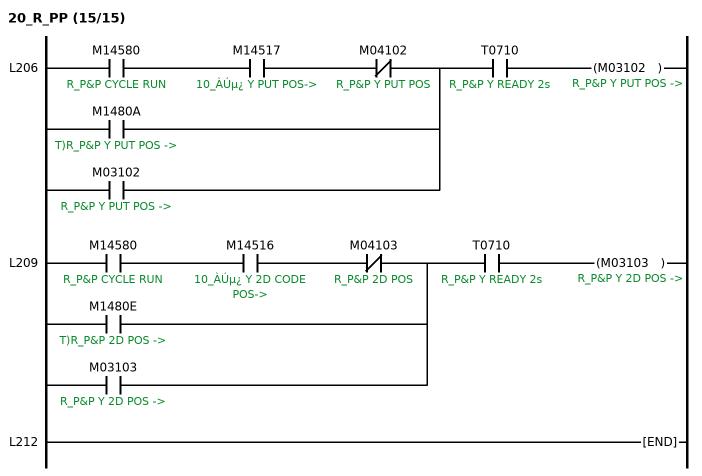
; L206
LOAD      M14580	// R_P&P CYCLE RUN
AND       M14517	// 10_ÀÚµ¿ Y PUT POS->
AND NOT   M04102	// R_P&P Y PUT POS
OR        M1480A	// T)R_P&P Y PUT POS ->
OR        M03102	// R_P&P Y PUT POS ->
AND       T0710	// R_P&P Y READY 2s
OUT       M03102	// R_P&P Y PUT POS ->
; L209
LOAD      M14580	// R_P&P CYCLE RUN
AND       M14516	// 10_ÀÚµ¿ Y 2D CODE POS->
AND NOT   M04103	// R_P&P 2D POS
OR        M1480E	// T)R_P&P 2D POS ->
OR        M03103	// R_P&P Y 2D POS ->
AND       T0710	// R_P&P Y READY 2s
OUT       M03103	// R_P&P Y 2D POS ->
; L212
END

PROGRAM 30_IN_LR_BUFFER (task: ½ºÄµ ÇÁ·Î±×·¥)

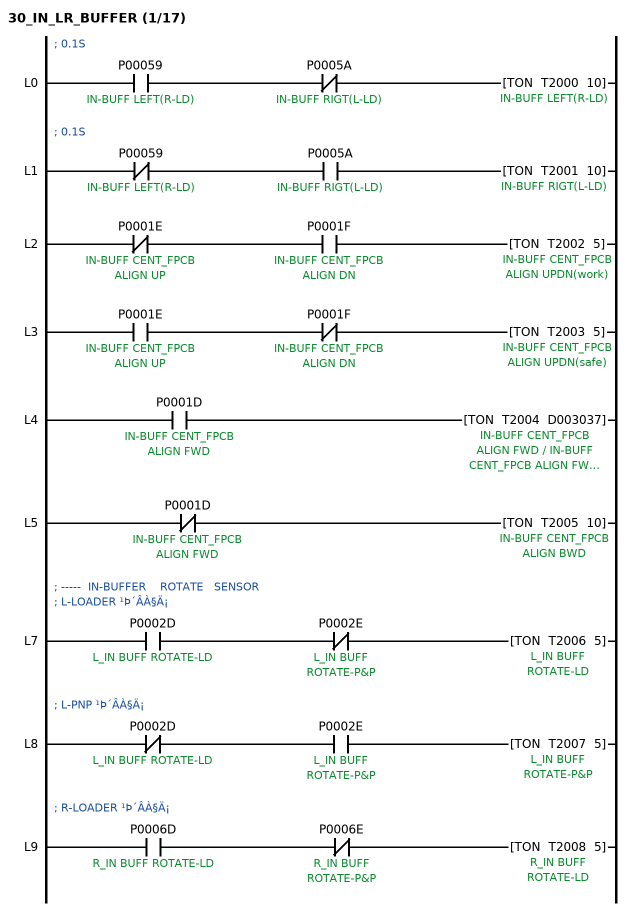
; L0
LOAD      P00059	// IN-BUFF LEFT(R-LD)
AND NOT   P0005A	// IN-BUFF RIGT(L-LD)
TON       T2000 10	// IN-BUFF LEFT(R-LD)
// output comment: 0.1S
; L1
LOAD NOT  P00059	// IN-BUFF LEFT(R-LD)
AND       P0005A	// IN-BUFF RIGT(L-LD)
TON       T2001 10	// IN-BUFF RIGT(L-LD)
// output comment: 0.1S
; L2
LOAD NOT  P0001E	// IN-BUFF CENT_FPCB ALIGN UP
AND       P0001F	// IN-BUFF CENT_FPCB ALIGN DN
TON       T2002 5	// IN-BUFF CENT_FPCB ALIGN UPDN(work)
; L3
LOAD      P0001E	// IN-BUFF CENT_FPCB ALIGN UP
AND NOT   P0001F	// IN-BUFF CENT_FPCB ALIGN DN
TON       T2003 5	// IN-BUFF CENT_FPCB ALIGN UPDN(safe)
; L4
LOAD      P0001D	// IN-BUFF CENT_FPCB ALIGN FWD
TON       T2004 D003037	// IN-BUFF CENT_FPCB ALIGN FWD / IN-BUFF CENT_FPCB ALIGN FWD DELAY
; L5
LOAD NOT  P0001D	// IN-BUFF CENT_FPCB ALIGN FWD
TON       T2005 10	// IN-BUFF CENT_FPCB ALIGN BWD
// -----  IN-BUFFER    ROTATE   SENSOR
; L7
LOAD      P0002D	// L_IN BUFF ROTATE-LD
AND NOT   P0002E	// L_IN BUFF ROTATE-P&P
TON       T2006 5	// L_IN BUFF ROTATE-LD
// output comment: L-LOADER ¹Þ´ÂÀ§Ä¡
; L8
LOAD NOT  P0002D	// L_IN BUFF ROTATE-LD
AND       P0002E	// L_IN BUFF ROTATE-P&P
TON       T2007 5	// L_IN BUFF ROTATE-P&P
// output comment: L-PNP ¹Þ´ÂÀ§Ä¡
; L9
LOAD      P0006D	// R_IN BUFF ROTATE-LD
AND NOT   P0006E	// R_IN BUFF ROTATE-P&P
TON       T2008 5	// R_IN BUFF ROTATE-LD
// output comment: R-LOADER ¹Þ´ÂÀ§Ä¡

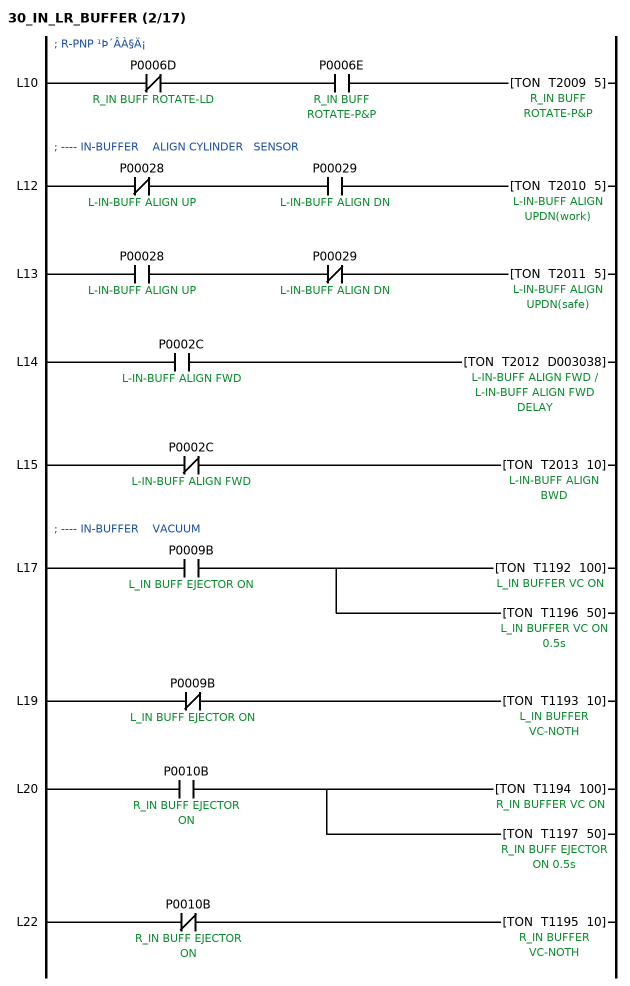
; L10
LOAD NOT  P0006D	// R_IN BUFF ROTATE-LD
AND       P0006E	// R_IN BUFF ROTATE-P&P
TON       T2009 5	// R_IN BUFF ROTATE-P&P
// output comment: R-PNP ¹Þ´ÂÀ§Ä¡
// ---- IN-BUFFER    ALIGN CYLINDER   SENSOR
; L12
LOAD NOT  P00028	// L-IN-BUFF ALIGN UP
AND       P00029	// L-IN-BUFF ALIGN DN
TON       T2010 5	// L-IN-BUFF ALIGN UPDN(work)
; L13
LOAD      P00028	// L-IN-BUFF ALIGN UP
AND NOT   P00029	// L-IN-BUFF ALIGN DN
TON       T2011 5	// L-IN-BUFF ALIGN UPDN(safe)
; L14
LOAD      P0002C	// L-IN-BUFF ALIGN FWD
TON       T2012 D003038	// L-IN-BUFF ALIGN FWD / L-IN-BUFF ALIGN FWD DELAY
; L15
LOAD NOT  P0002C	// L-IN-BUFF ALIGN FWD
TON       T2013 10	// L-IN-BUFF ALIGN BWD
// ---- IN-BUFFER    VACUUM
; L17
LOAD      P0009B	// L_IN BUFF EJECTOR ON
TON       T1192 100	// L_IN BUFFER VC ON
TON       T1196 50	// L_IN BUFFER VC ON 0.5s
; L19
LOAD NOT  P0009B	// L_IN BUFF EJECTOR ON
TON       T1193 10	// L_IN BUFFER VC-NOTH
; L20
LOAD      P0010B	// R_IN BUFF EJECTOR ON
TON       T1194 100	// R_IN BUFFER VC ON
TON       T1197 50	// R_IN BUFF EJECTOR ON 0.5s
; L22
LOAD NOT  P0010B	// R_IN BUFF EJECTOR ON
TON       T1195 10	// R_IN BUFFER VC-NOTH

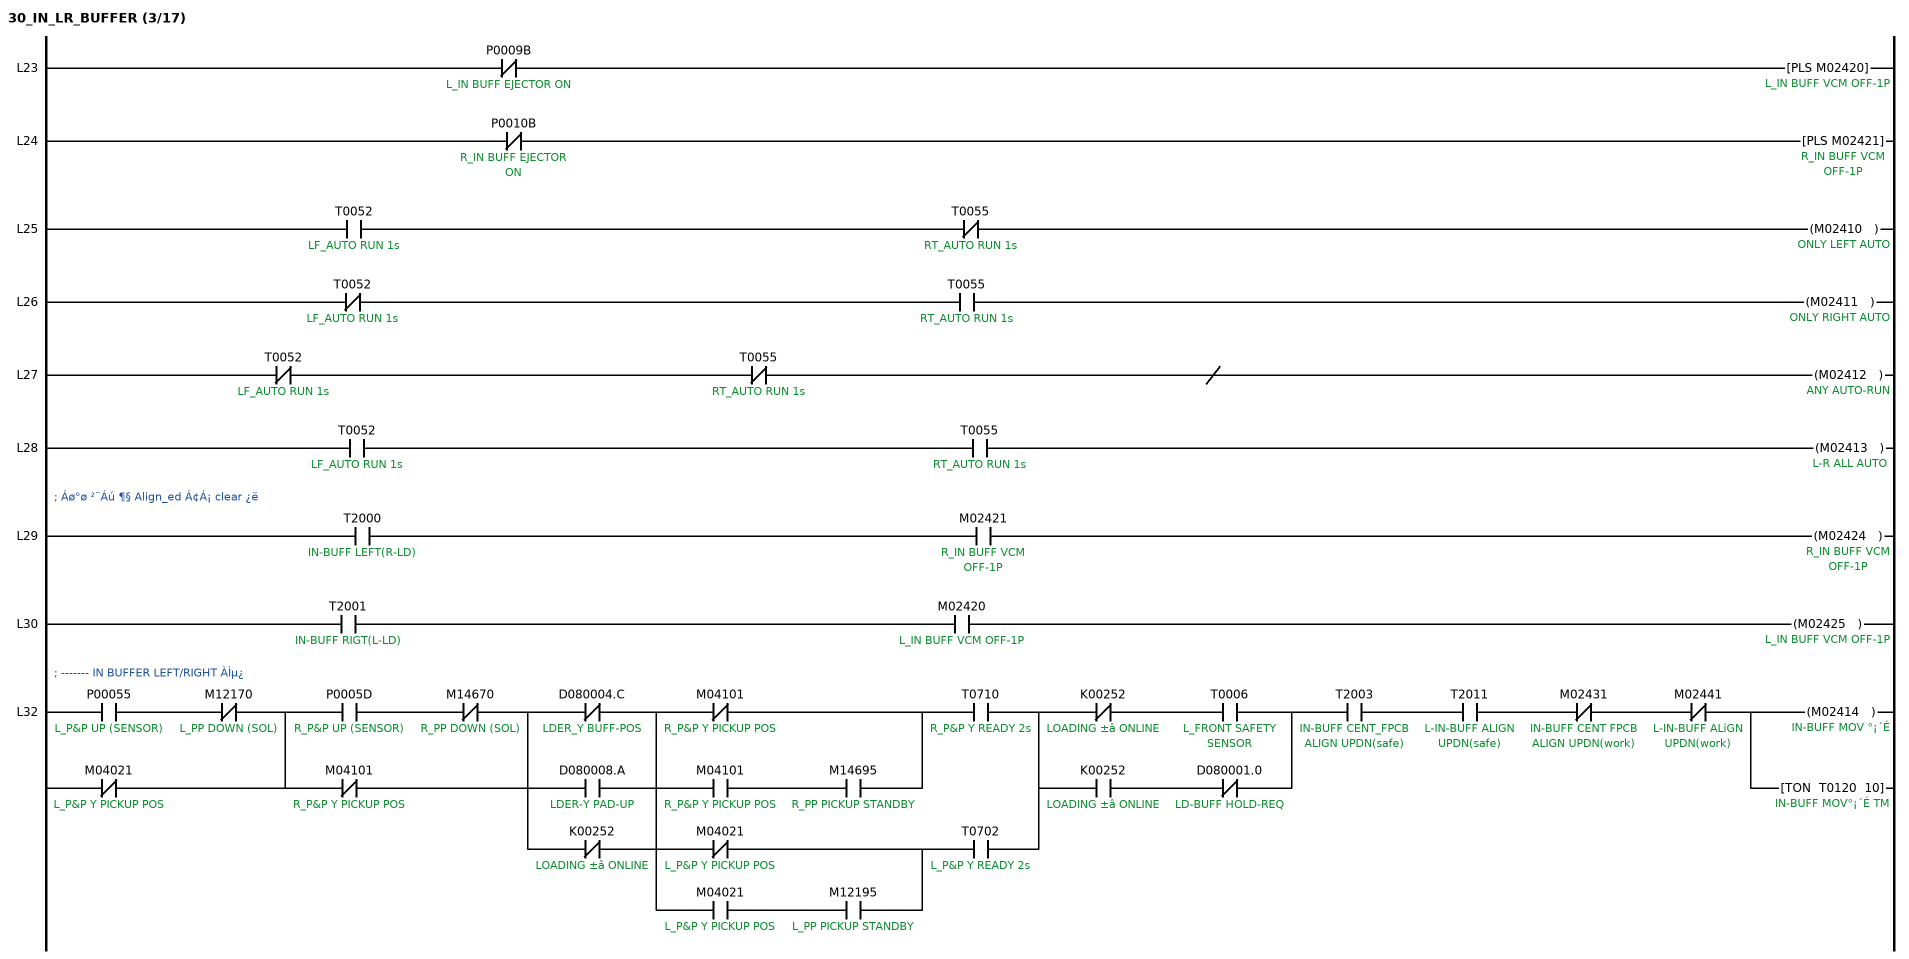
; L23
LOAD NOT  P0009B	// L_IN BUFF EJECTOR ON
OUTP      M02420	// L_IN BUFF VCM OFF-1P
; L24
LOAD NOT  P0010B	// R_IN BUFF EJECTOR ON
OUTP      M02421	// R_IN BUFF VCM OFF-1P
; L25
LOAD      T0052	// LF_AUTO RUN 1s
AND NOT   T0055	// RT_AUTO RUN 1s
OUT       M02410	// ONLY LEFT AUTO
; L26
LOAD NOT  T0052	// LF_AUTO RUN 1s
AND       T0055	// RT_AUTO RUN 1s
OUT       M02411	// ONLY RIGHT AUTO
; L27
LOAD NOT  T0052	// LF_AUTO RUN 1s
AND NOT   T0055	// RT_AUTO RUN 1s
NOT
OUT       M02412	// ANY AUTO-RUN
; L28
LOAD      T0052	// LF_AUTO RUN 1s
AND       T0055	// RT_AUTO RUN 1s
OUT       M02413	// L-R ALL AUTO
; L29
LOAD      T2000	// IN-BUFF LEFT(R-LD)
AND       M02421	// R_IN BUFF VCM OFF-1P
OUT       M02424	// R_IN BUFF VCM OFF-1P
// output comment: Áø°ø ²¨Áú ¶§ Align_ed Á¢Á¡ clear ¿ë
; L30
LOAD      T2001	// IN-BUFF RIGT(L-LD)
AND       M02420	// L_IN BUFF VCM OFF-1P
OUT       M02425	// L_IN BUFF VCM OFF-1P
// ------- IN BUFFER LEFT/RIGHT ÀÌµ¿
; L32
LOAD      P00055	// L_P&P UP (SENSOR)
AND NOT   M12170	// L_PP DOWN (SOL)
OR NOT    M04021	// L_P&P Y PICKUP POS
LOAD      P0005D	// R_P&P UP (SENSOR)
AND NOT   M14670	// R_PP DOWN (SOL)
OR NOT    M04101	// R_P&P Y PICKUP POS
AND LOAD
LOAD NOT  D080004.C	// LDER_Y BUFF-POS
OR        D080008.A	// LDER-Y PAD-UP
OR NOT    K00252	// LOADING ±â ONLINE
AND LOAD
LOAD NOT  M04101	// R_P&P Y PICKUP POS
LOAD      M04101	// R_P&P Y PICKUP POS
AND       M14695	// R_PP PICKUP STANDBY
OR LOAD
AND       T0710	// R_P&P Y READY 2s
LOAD NOT  M04021	// L_P&P Y PICKUP POS
LOAD      M04021	// L_P&P Y PICKUP POS
AND       M12195	// L_PP PICKUP STANDBY
OR LOAD
AND       T0702	// L_P&P Y READY 2s
OR LOAD
AND LOAD
LOAD NOT  K00252	// LOADING ±â ONLINE
AND       T0006	// L_FRONT SAFETY SENSOR
LOAD      K00252	// LOADING ±â ONLINE
AND NOT   D080001.0	// LD-BUFF HOLD-REQ
OR LOAD
AND LOAD
AND       T2003	// IN-BUFF CENT_FPCB ALIGN UPDN(safe)
AND       T2011	// L-IN-BUFF ALIGN UPDN(safe)
AND NOT   M02431	// IN-BUFF CENT FPCB ALIGN UPDN(work)
AND NOT   M02441	// L-IN-BUFF ALiGN UPDN(work)
OUT       M02414	// IN-BUFF MOV °¡´É
TON       T0120 10	// IN-BUFF MOV°¡´É TM

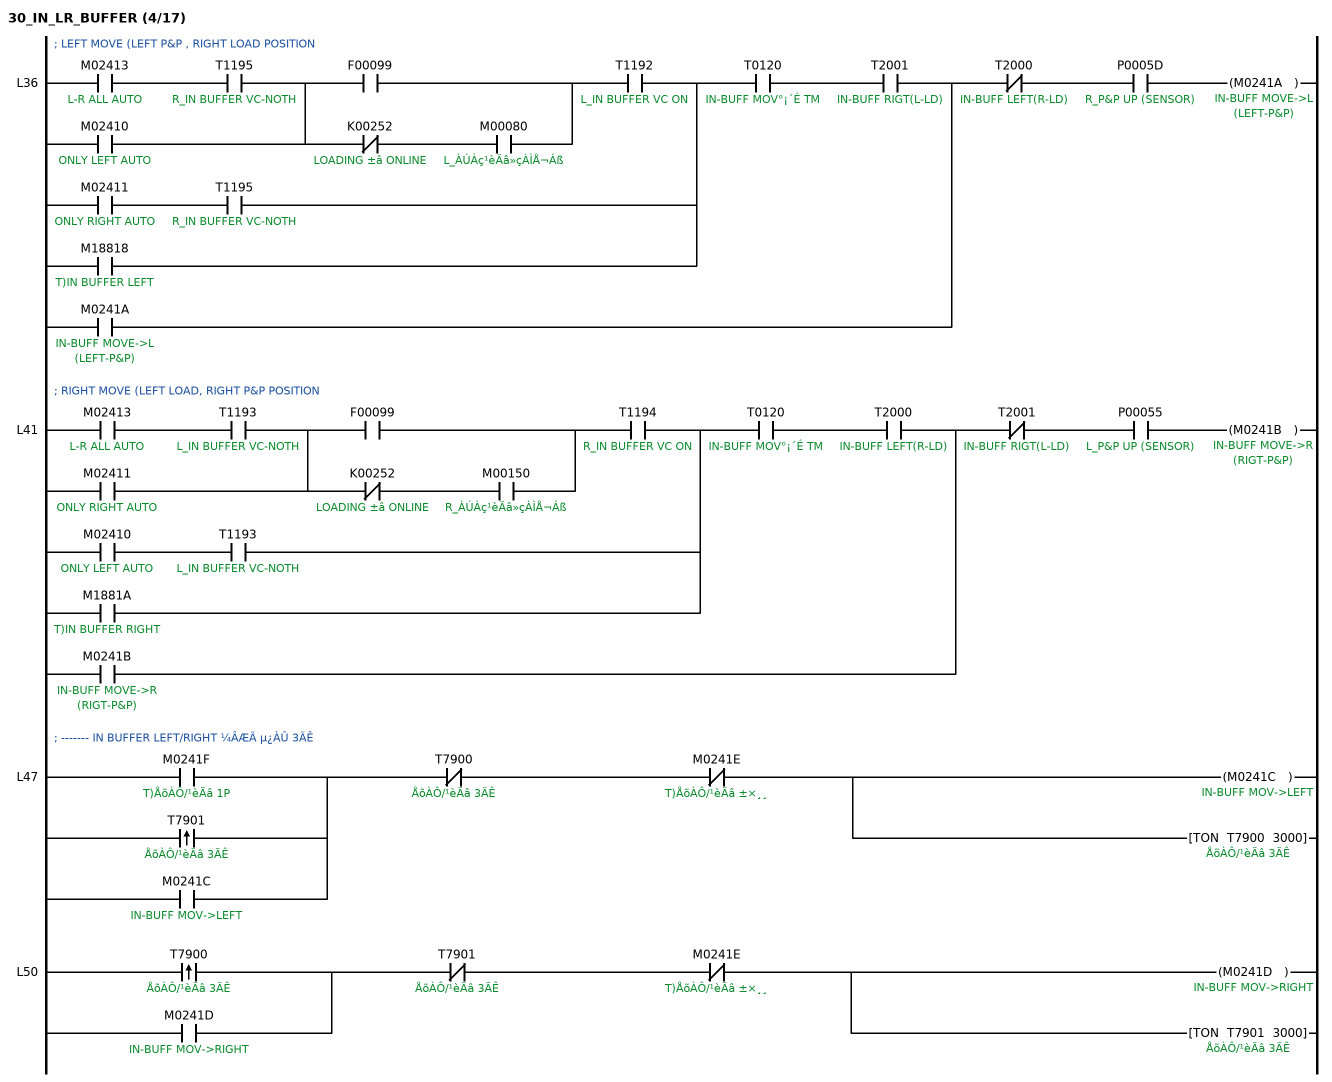
; L36
LOAD      M02413	// L-R ALL AUTO
AND       T1195	// R_IN BUFFER VC-NOTH
OR        M02410	// ONLY LEFT AUTO
LOAD      F00099
LOAD NOT  K00252	// LOADING ±â ONLINE
AND       M00080	// L_ÀÚÀç¹èÃâ»çÀÌÅ¬Áß
OR LOAD
AND LOAD
AND       T1192	// L_IN BUFFER VC ON
LOAD      M02411	// ONLY RIGHT AUTO
AND       T1195	// R_IN BUFFER VC-NOTH
OR LOAD
OR        M18818	// T)IN BUFFER LEFT
AND       T0120	// IN-BUFF MOV°¡´É TM
AND       T2001	// IN-BUFF RIGT(L-LD)
OR        M0241A	// IN-BUFF MOVE->L (LEFT-P&P)
AND NOT   T2000	// IN-BUFF LEFT(R-LD)
AND       P0005D	// R_P&P UP (SENSOR)
OUT       M0241A	// IN-BUFF MOVE->L (LEFT-P&P)
// output comment: LEFT MOVE (LEFT P&P , RIGHT LOAD POSITION
; L41
LOAD      M02413	// L-R ALL AUTO
AND       T1193	// L_IN BUFFER VC-NOTH
OR        M02411	// ONLY RIGHT AUTO
LOAD      F00099
LOAD NOT  K00252	// LOADING ±â ONLINE
AND       M00150	// R_ÀÚÀç¹èÃâ»çÀÌÅ¬Áß
OR LOAD
AND LOAD
AND       T1194	// R_IN BUFFER VC ON
LOAD      M02410	// ONLY LEFT AUTO
AND       T1193	// L_IN BUFFER VC-NOTH
OR LOAD
OR        M1881A	// T)IN BUFFER RIGHT
AND       T0120	// IN-BUFF MOV°¡´É TM
AND       T2000	// IN-BUFF LEFT(R-LD)
OR        M0241B	// IN-BUFF MOVE->R (RIGT-P&P)
AND NOT   T2001	// IN-BUFF RIGT(L-LD)
AND       P00055	// L_P&P UP (SENSOR)
OUT       M0241B	// IN-BUFF MOVE->R (RIGT-P&P)
// output comment: RIGHT MOVE (LEFT LOAD, RIGHT P&P POSITION
// ------- IN BUFFER LEFT/RIGHT ¼ÂÆÃ µ¿ÀÛ 3ÃÊ
; L47
LOAD      M0241F	// T)ÅõÀÔ/¹èÃâ 1P
ORP       T7901	// ÅõÀÔ/¹èÃâ 3ÃÊ
OR        M0241C	// IN-BUFF MOV->LEFT
AND NOT   T7900	// ÅõÀÔ/¹èÃâ 3ÃÊ
AND NOT   M0241E	// T)ÅõÀÔ/¹èÃâ ±×¸¸
OUT       M0241C	// IN-BUFF MOV->LEFT
TON       T7900 3000	// ÅõÀÔ/¹èÃâ 3ÃÊ
; L50
LOADP     T7900	// ÅõÀÔ/¹èÃâ 3ÃÊ
OR        M0241D	// IN-BUFF MOV->RIGHT
AND NOT   T7901	// ÅõÀÔ/¹èÃâ 3ÃÊ
AND NOT   M0241E	// T)ÅõÀÔ/¹èÃâ ±×¸¸
OUT       M0241D	// IN-BUFF MOV->RIGHT
TON       T7901 3000	// ÅõÀÔ/¹èÃâ 3ÃÊ

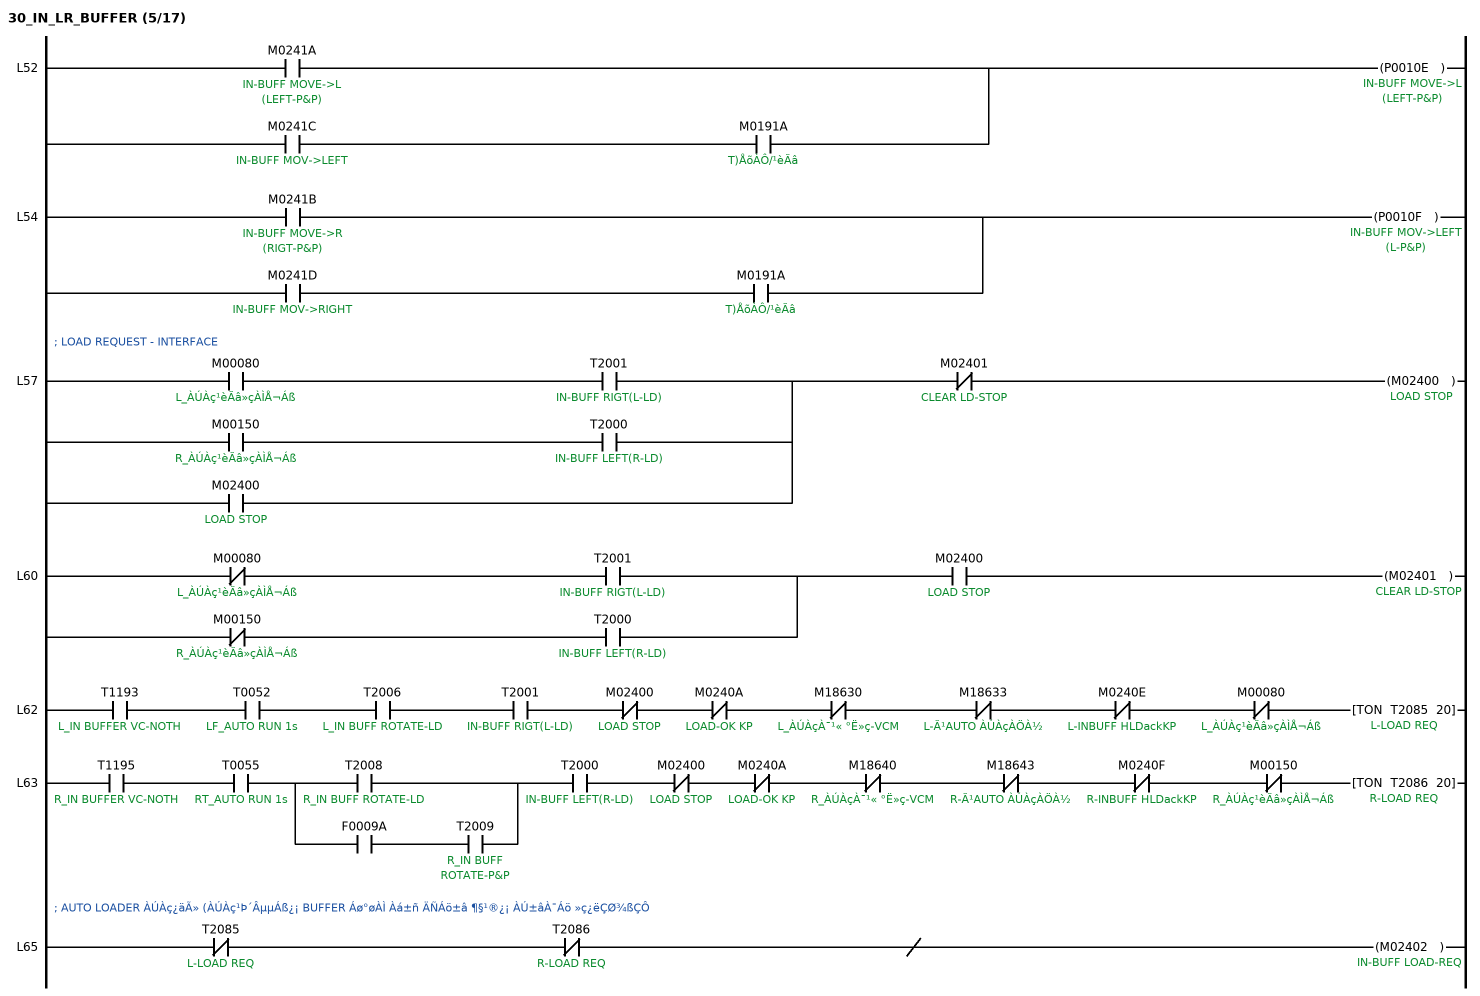
; L52
LOAD      M0241A	// IN-BUFF MOVE->L (LEFT-P&P)
LOAD      M0241C	// IN-BUFF MOV->LEFT
AND       M0191A	// T)ÅõÀÔ/¹èÃâ
OR LOAD
OUT       P0010E	// IN-BUFF MOVE->L (LEFT-P&P)
; L54
LOAD      M0241B	// IN-BUFF MOVE->R (RIGT-P&P)
LOAD      M0241D	// IN-BUFF MOV->RIGHT
AND       M0191A	// T)ÅõÀÔ/¹èÃâ
OR LOAD
OUT       P0010F	// IN-BUFF MOV->LEFT (L-P&P)
// LOAD REQUEST - INTERFACE
; L57
LOAD      M00080	// L_ÀÚÀç¹èÃâ»çÀÌÅ¬Áß
AND       T2001	// IN-BUFF RIGT(L-LD)
LOAD      M00150	// R_ÀÚÀç¹èÃâ»çÀÌÅ¬Áß
AND       T2000	// IN-BUFF LEFT(R-LD)
OR LOAD
OR        M02400	// LOAD STOP
AND NOT   M02401	// CLEAR LD-STOP
OUT       M02400	// LOAD STOP
; L60
LOAD NOT  M00080	// L_ÀÚÀç¹èÃâ»çÀÌÅ¬Áß
AND       T2001	// IN-BUFF RIGT(L-LD)
LOAD NOT  M00150	// R_ÀÚÀç¹èÃâ»çÀÌÅ¬Áß
AND       T2000	// IN-BUFF LEFT(R-LD)
OR LOAD
AND       M02400	// LOAD STOP
OUT       M02401	// CLEAR LD-STOP
; L62
LOAD      T1193	// L_IN BUFFER VC-NOTH
AND       T0052	// LF_AUTO RUN 1s
AND       T2006	// L_IN BUFF ROTATE-LD
AND       T2001	// IN-BUFF RIGT(L-LD)
AND NOT   M02400	// LOAD STOP
AND NOT   M0240A	// LOAD-OK KP
AND NOT   M18630	// L_ÀÚÀçÀ¯¹« °Ë»ç-VCM
AND NOT   M18633	// L-Ã¹AUTO ÀÚÀçÀÖÀ½
AND NOT   M0240E	// L-INBUFF HLDackKP
AND NOT   M00080	// L_ÀÚÀç¹èÃâ»çÀÌÅ¬Áß
TON       T2085 20	// L-LOAD REQ
; L63
LOAD      T1195	// R_IN BUFFER VC-NOTH
AND       T0055	// RT_AUTO RUN 1s
LOAD      T2008	// R_IN BUFF ROTATE-LD
LOAD      F0009A
AND       T2009	// R_IN BUFF ROTATE-P&P
OR LOAD
AND LOAD
AND       T2000	// IN-BUFF LEFT(R-LD)
AND NOT   M02400	// LOAD STOP
AND NOT   M0240A	// LOAD-OK KP
AND NOT   M18640	// R_ÀÚÀçÀ¯¹« °Ë»ç-VCM
AND NOT   M18643	// R-Ã¹AUTO ÀÚÀçÀÖÀ½
AND NOT   M0240F	// R-INBUFF HLDackKP
AND NOT   M00150	// R_ÀÚÀç¹èÃâ»çÀÌÅ¬Áß
TON       T2086 20	// R-LOAD REQ
; L65
LOAD NOT  T2085	// L-LOAD REQ
AND NOT   T2086	// R-LOAD REQ
NOT
OUT       M02402	// IN-BUFF LOAD-REQ
// output comment: AUTO LOADER ÀÚÀç¿äÃ» (ÀÚÀç¹Þ´ÂµµÁß¿¡ BUFFER Áø°øÀÌ Àá±ñ ÄÑÁö±â ¶§¹®¿¡ ÀÚ±âÀ¯Áö »ç¿ëÇØ¾ßÇÔ

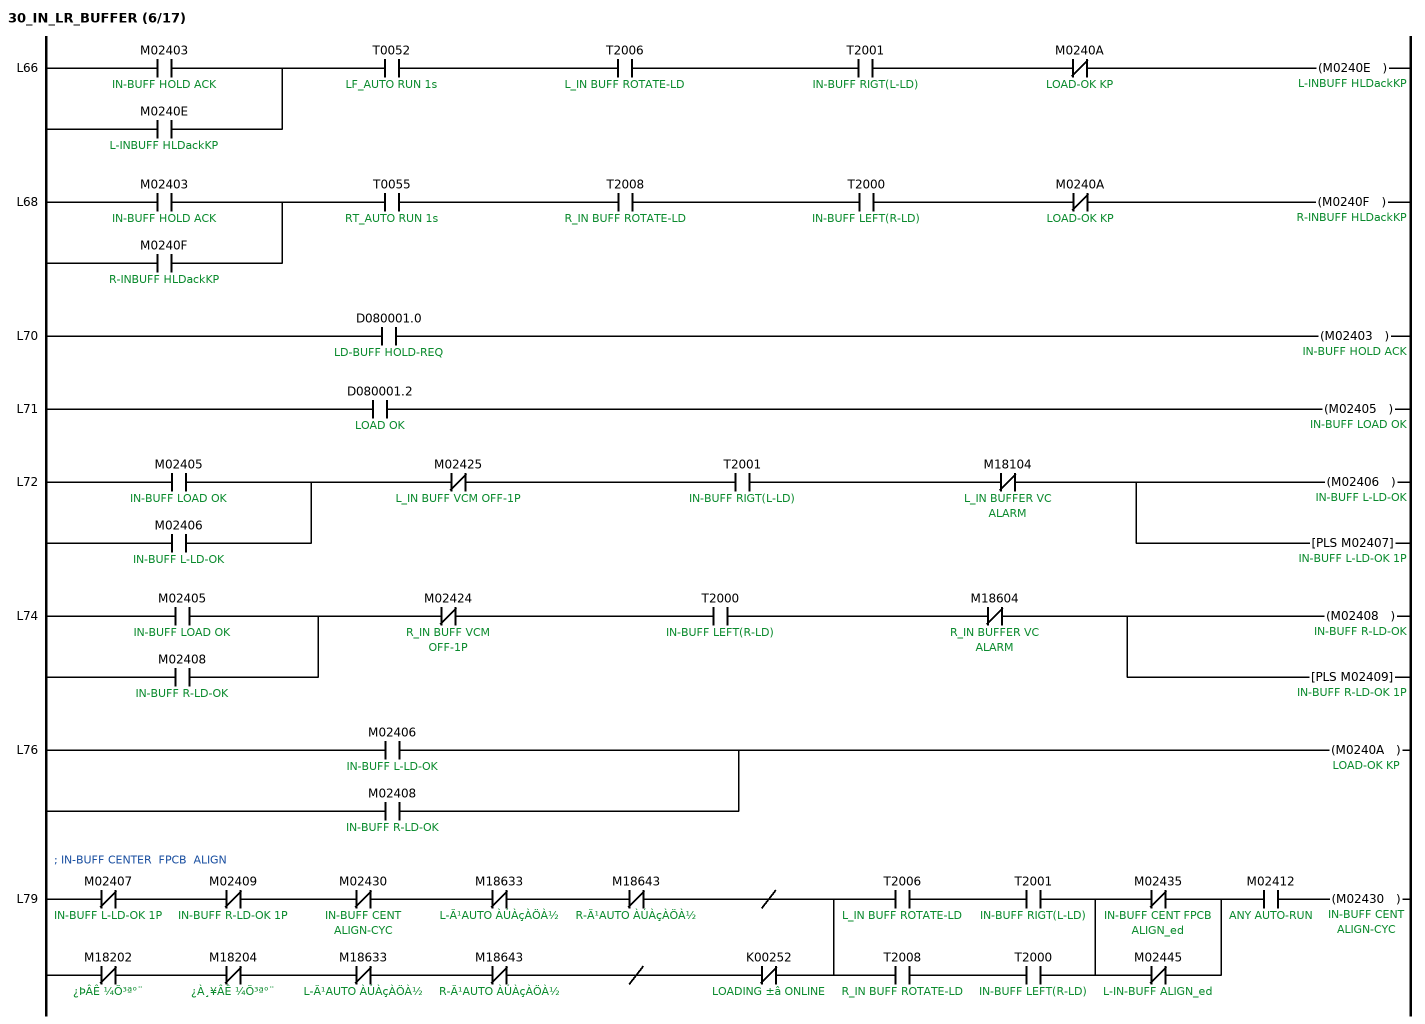
; L66
LOAD      M02403	// IN-BUFF HOLD ACK
OR        M0240E	// L-INBUFF HLDackKP
AND       T0052	// LF_AUTO RUN 1s
AND       T2006	// L_IN BUFF ROTATE-LD
AND       T2001	// IN-BUFF RIGT(L-LD)
AND NOT   M0240A	// LOAD-OK KP
OUT       M0240E	// L-INBUFF HLDackKP
; L68
LOAD      M02403	// IN-BUFF HOLD ACK
OR        M0240F	// R-INBUFF HLDackKP
AND       T0055	// RT_AUTO RUN 1s
AND       T2008	// R_IN BUFF ROTATE-LD
AND       T2000	// IN-BUFF LEFT(R-LD)
AND NOT   M0240A	// LOAD-OK KP
OUT       M0240F	// R-INBUFF HLDackKP
; L70
LOAD      D080001.0	// LD-BUFF HOLD-REQ
OUT       M02403	// IN-BUFF HOLD ACK
; L71
LOAD      D080001.2	// LOAD OK
OUT       M02405	// IN-BUFF LOAD OK
; L72
LOAD      M02405	// IN-BUFF LOAD OK
OR        M02406	// IN-BUFF L-LD-OK
AND NOT   M02425	// L_IN BUFF VCM OFF-1P
AND       T2001	// IN-BUFF RIGT(L-LD)
AND NOT   M18104	// L_IN BUFFER VC ALARM
OUT       M02406	// IN-BUFF L-LD-OK
OUTP      M02407	// IN-BUFF L-LD-OK 1P
; L74
LOAD      M02405	// IN-BUFF LOAD OK
OR        M02408	// IN-BUFF R-LD-OK
AND NOT   M02424	// R_IN BUFF VCM OFF-1P
AND       T2000	// IN-BUFF LEFT(R-LD)
AND NOT   M18604	// R_IN BUFFER VC ALARM
OUT       M02408	// IN-BUFF R-LD-OK
OUTP      M02409	// IN-BUFF R-LD-OK 1P
; L76
LOAD      M02406	// IN-BUFF L-LD-OK
OR        M02408	// IN-BUFF R-LD-OK
OUT       M0240A	// LOAD-OK KP
// IN-BUFF CENTER  FPCB  ALIGN
; L79
LOAD NOT  M02407	// IN-BUFF L-LD-OK 1P
AND NOT   M02409	// IN-BUFF R-LD-OK 1P
AND NOT   M02430	// IN-BUFF CENT ALIGN-CYC
AND NOT   M18633	// L-Ã¹AUTO ÀÚÀçÀÖÀ½
AND NOT   M18643	// R-Ã¹AUTO ÀÚÀçÀÖÀ½
NOT
LOAD NOT  M18202	// ¿ÞÂÊ ¼Õ³ª°¨
AND NOT   M18204	// ¿À¸¥ÂÊ ¼Õ³ª°¨
AND NOT   M18633	// L-Ã¹AUTO ÀÚÀçÀÖÀ½
AND NOT   M18643	// R-Ã¹AUTO ÀÚÀçÀÖÀ½
NOT
AND NOT   K00252	// LOADING ±â ONLINE
OR LOAD
LOAD      T2006	// L_IN BUFF ROTATE-LD
AND       T2001	// IN-BUFF RIGT(L-LD)
LOAD      T2008	// R_IN BUFF ROTATE-LD
AND       T2000	// IN-BUFF LEFT(R-LD)
OR LOAD
AND LOAD
LOAD NOT  M02435	// IN-BUFF CENT FPCB ALIGN_ed
OR NOT    M02445	// L-IN-BUFF ALIGN_ed
AND LOAD
AND       M02412	// ANY AUTO-RUN
OUT       M02430	// IN-BUFF CENT ALIGN-CYC

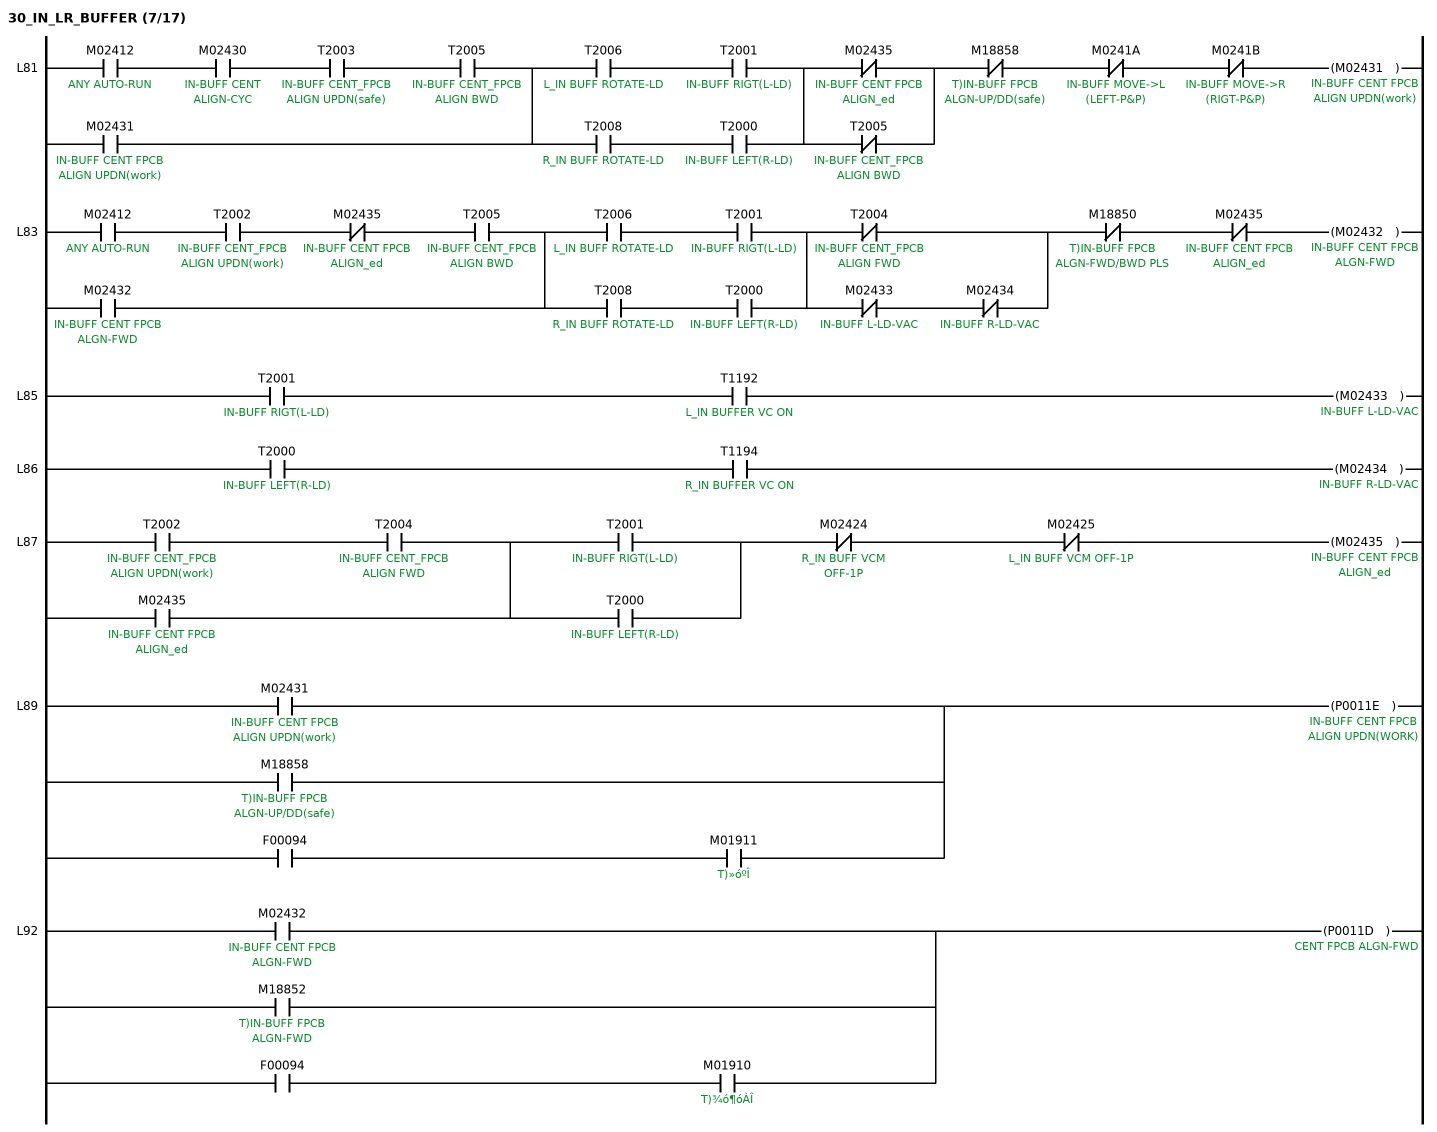
; L81
LOAD      M02412	// ANY AUTO-RUN
AND       M02430	// IN-BUFF CENT ALIGN-CYC
AND       T2003	// IN-BUFF CENT_FPCB ALIGN UPDN(safe)
AND       T2005	// IN-BUFF CENT_FPCB ALIGN BWD
OR        M02431	// IN-BUFF CENT FPCB ALIGN UPDN(work)
LOAD      T2006	// L_IN BUFF ROTATE-LD
AND       T2001	// IN-BUFF RIGT(L-LD)
LOAD      T2008	// R_IN BUFF ROTATE-LD
AND       T2000	// IN-BUFF LEFT(R-LD)
OR LOAD
AND LOAD
LOAD NOT  M02435	// IN-BUFF CENT FPCB ALIGN_ed
OR NOT    T2005	// IN-BUFF CENT_FPCB ALIGN BWD
AND LOAD
AND NOT   M18858	// T)IN-BUFF FPCB ALGN-UP/DD(safe)
AND NOT   M0241A	// IN-BUFF MOVE->L (LEFT-P&P)
AND NOT   M0241B	// IN-BUFF MOVE->R (RIGT-P&P)
OUT       M02431	// IN-BUFF CENT FPCB ALIGN UPDN(work)
; L83
LOAD      M02412	// ANY AUTO-RUN
AND       T2002	// IN-BUFF CENT_FPCB ALIGN UPDN(work)
AND NOT   M02435	// IN-BUFF CENT FPCB ALIGN_ed
AND       T2005	// IN-BUFF CENT_FPCB ALIGN BWD
OR        M02432	// IN-BUFF CENT FPCB ALGN-FWD
LOAD      T2006	// L_IN BUFF ROTATE-LD
AND       T2001	// IN-BUFF RIGT(L-LD)
LOAD      T2008	// R_IN BUFF ROTATE-LD
AND       T2000	// IN-BUFF LEFT(R-LD)
OR LOAD
AND LOAD
LOAD NOT  T2004	// IN-BUFF CENT_FPCB ALIGN FWD
LOAD NOT  M02433	// IN-BUFF L-LD-VAC
AND NOT   M02434	// IN-BUFF R-LD-VAC
OR LOAD
AND LOAD
AND NOT   M18850	// T)IN-BUFF FPCB ALGN-FWD/BWD PLS
AND NOT   M02435	// IN-BUFF CENT FPCB ALIGN_ed
OUT       M02432	// IN-BUFF CENT FPCB ALGN-FWD
; L85
LOAD      T2001	// IN-BUFF RIGT(L-LD)
AND       T1192	// L_IN BUFFER VC ON
OUT       M02433	// IN-BUFF L-LD-VAC
; L86
LOAD      T2000	// IN-BUFF LEFT(R-LD)
AND       T1194	// R_IN BUFFER VC ON
OUT       M02434	// IN-BUFF R-LD-VAC
; L87
LOAD      T2002	// IN-BUFF CENT_FPCB ALIGN UPDN(work)
AND       T2004	// IN-BUFF CENT_FPCB ALIGN FWD
OR        M02435	// IN-BUFF CENT FPCB ALIGN_ed
LOAD      T2001	// IN-BUFF RIGT(L-LD)
OR        T2000	// IN-BUFF LEFT(R-LD)
AND LOAD
AND NOT   M02424	// R_IN BUFF VCM OFF-1P
AND NOT   M02425	// L_IN BUFF VCM OFF-1P
OUT       M02435	// IN-BUFF CENT FPCB ALIGN_ed
; L89
LOAD      M02431	// IN-BUFF CENT FPCB ALIGN UPDN(work)
OR        M18858	// T)IN-BUFF FPCB ALGN-UP/DD(safe)
LOAD      F00094
AND       M01911	// T)»óºÎ
OR LOAD
OUT       P0011E	// IN-BUFF CENT FPCB ALIGN UPDN(WORK)
; L92
LOAD      M02432	// IN-BUFF CENT FPCB ALGN-FWD
OR        M18852	// T)IN-BUFF FPCB ALGN-FWD
LOAD      F00094
AND       M01910	// T)¾ó¶óÀÎ
OR LOAD
OUT       P0011D	// CENT FPCB ALGN-FWD

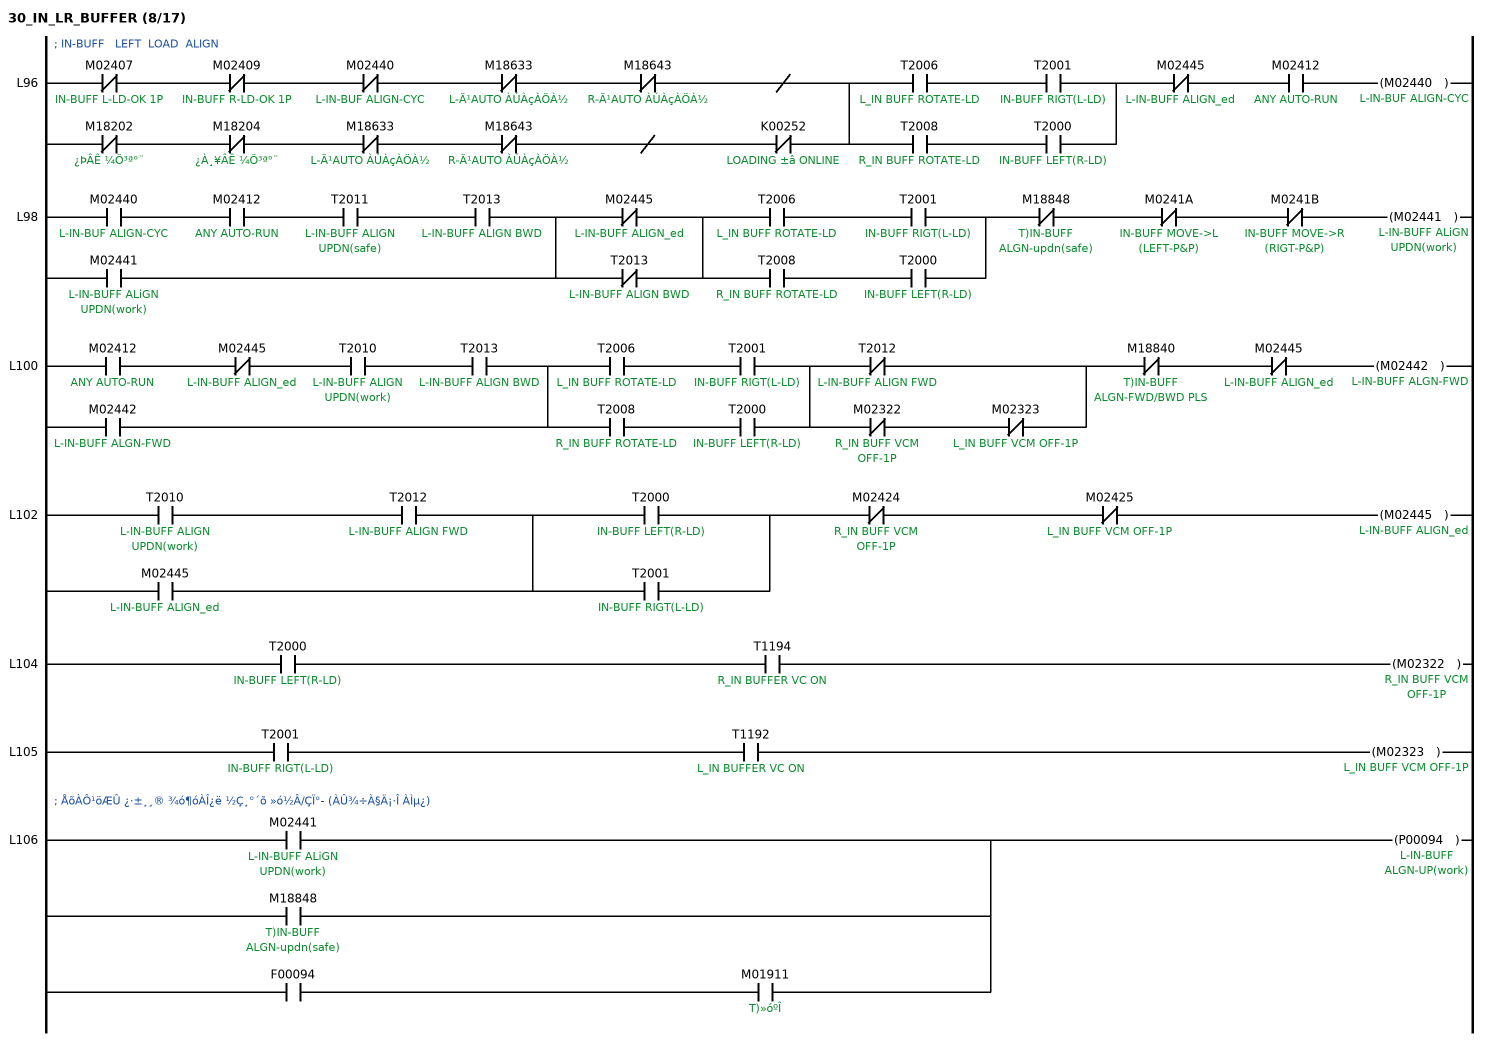
// IN-BUFF   LEFT  LOAD  ALIGN
; L96
LOAD NOT  M02407	// IN-BUFF L-LD-OK 1P
AND NOT   M02409	// IN-BUFF R-LD-OK 1P
AND NOT   M02440	// L-IN-BUF ALIGN-CYC
AND NOT   M18633	// L-Ã¹AUTO ÀÚÀçÀÖÀ½
AND NOT   M18643	// R-Ã¹AUTO ÀÚÀçÀÖÀ½
NOT
LOAD NOT  M18202	// ¿ÞÂÊ ¼Õ³ª°¨
AND NOT   M18204	// ¿À¸¥ÂÊ ¼Õ³ª°¨
AND NOT   M18633	// L-Ã¹AUTO ÀÚÀçÀÖÀ½
AND NOT   M18643	// R-Ã¹AUTO ÀÚÀçÀÖÀ½
NOT
AND NOT   K00252	// LOADING ±â ONLINE
OR LOAD
LOAD      T2006	// L_IN BUFF ROTATE-LD
AND       T2001	// IN-BUFF RIGT(L-LD)
LOAD      T2008	// R_IN BUFF ROTATE-LD
AND       T2000	// IN-BUFF LEFT(R-LD)
OR LOAD
AND LOAD
AND NOT   M02445	// L-IN-BUFF ALIGN_ed
AND       M02412	// ANY AUTO-RUN
OUT       M02440	// L-IN-BUF ALIGN-CYC
; L98
LOAD      M02440	// L-IN-BUF ALIGN-CYC
AND       M02412	// ANY AUTO-RUN
AND       T2011	// L-IN-BUFF ALIGN UPDN(safe)
AND       T2013	// L-IN-BUFF ALIGN BWD
OR        M02441	// L-IN-BUFF ALiGN UPDN(work)
LOAD NOT  M02445	// L-IN-BUFF ALIGN_ed
OR NOT    T2013	// L-IN-BUFF ALIGN BWD
AND LOAD
LOAD      T2006	// L_IN BUFF ROTATE-LD
AND       T2001	// IN-BUFF RIGT(L-LD)
LOAD      T2008	// R_IN BUFF ROTATE-LD
AND       T2000	// IN-BUFF LEFT(R-LD)
OR LOAD
AND LOAD
AND NOT   M18848	// T)IN-BUFF ALGN-updn(safe)
AND NOT   M0241A	// IN-BUFF MOVE->L (LEFT-P&P)
AND NOT   M0241B	// IN-BUFF MOVE->R (RIGT-P&P)
OUT       M02441	// L-IN-BUFF ALiGN UPDN(work)
; L100
LOAD      M02412	// ANY AUTO-RUN
AND NOT   M02445	// L-IN-BUFF ALIGN_ed
AND       T2010	// L-IN-BUFF ALIGN UPDN(work)
AND       T2013	// L-IN-BUFF ALIGN BWD
OR        M02442	// L-IN-BUFF ALGN-FWD
LOAD      T2006	// L_IN BUFF ROTATE-LD
AND       T2001	// IN-BUFF RIGT(L-LD)
LOAD      T2008	// R_IN BUFF ROTATE-LD
AND       T2000	// IN-BUFF LEFT(R-LD)
OR LOAD
AND LOAD
LOAD NOT  T2012	// L-IN-BUFF ALIGN FWD
LOAD NOT  M02322	// R_IN BUFF VCM OFF-1P
AND NOT   M02323	// L_IN BUFF VCM OFF-1P
OR LOAD
AND LOAD
AND NOT   M18840	// T)IN-BUFF ALGN-FWD/BWD PLS
AND NOT   M02445	// L-IN-BUFF ALIGN_ed
OUT       M02442	// L-IN-BUFF ALGN-FWD
; L102
LOAD      T2010	// L-IN-BUFF ALIGN UPDN(work)
AND       T2012	// L-IN-BUFF ALIGN FWD
OR        M02445	// L-IN-BUFF ALIGN_ed
LOAD      T2000	// IN-BUFF LEFT(R-LD)
OR        T2001	// IN-BUFF RIGT(L-LD)
AND LOAD
AND NOT   M02424	// R_IN BUFF VCM OFF-1P
AND NOT   M02425	// L_IN BUFF VCM OFF-1P
OUT       M02445	// L-IN-BUFF ALIGN_ed
; L104
LOAD      T2000	// IN-BUFF LEFT(R-LD)
AND       T1194	// R_IN BUFFER VC ON
OUT       M02322	// R_IN BUFF VCM OFF-1P
; L105
LOAD      T2001	// IN-BUFF RIGT(L-LD)
AND       T1192	// L_IN BUFFER VC ON
OUT       M02323	// L_IN BUFF VCM OFF-1P
; L106
LOAD      M02441	// L-IN-BUFF ALiGN UPDN(work)
OR        M18848	// T)IN-BUFF ALGN-updn(safe)
LOAD      F00094
AND       M01911	// T)»óºÎ
OR LOAD
OUT       P00094	// L-IN-BUFF ALGN-UP(work)
// output comment: ÅõÀÔ¹öÆÛ ¿·±¸¸® ¾ó¶óÀÎ¿ë ½Ç¸°´õ »ó½Â/ÇÏ°­ (ÀÛ¾÷À§Ä¡·Î ÀÌµ¿)

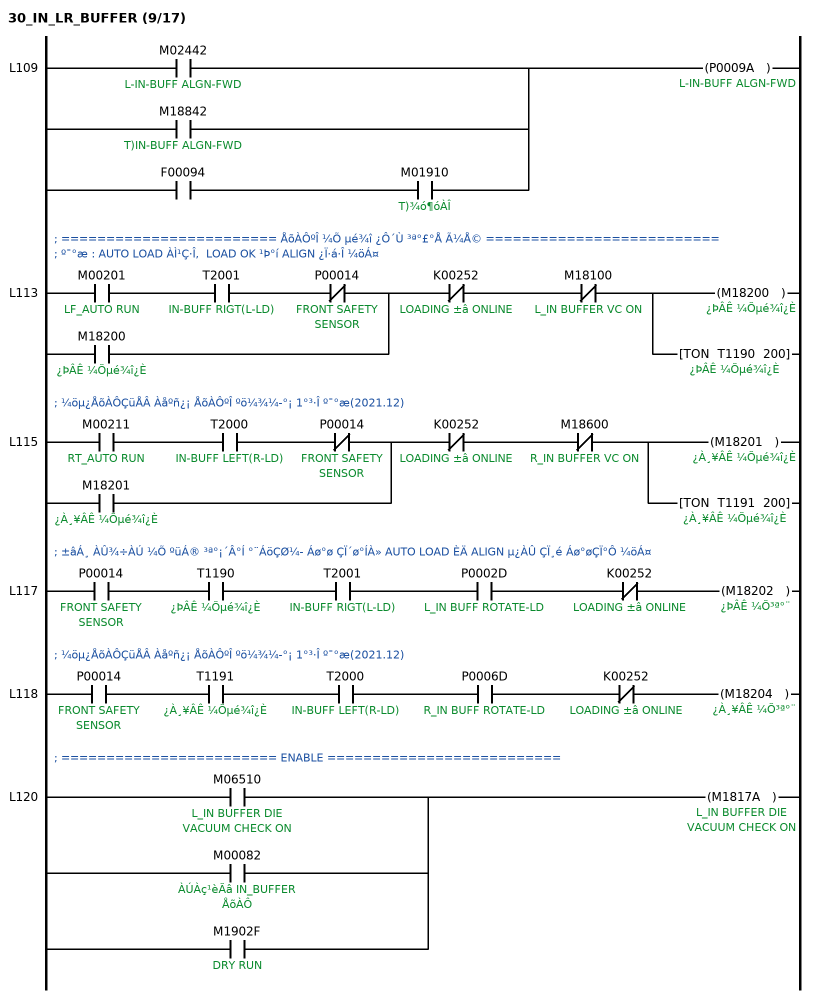
; L109
LOAD      M02442	// L-IN-BUFF ALGN-FWD
OR        M18842	// T)IN-BUFF ALGN-FWD
LOAD      F00094
AND       M01910	// T)¾ó¶óÀÎ
OR LOAD
OUT       P0009A	// L-IN-BUFF ALGN-FWD
// ======================== ÅõÀÔºÎ ¼Õ µé¾î ¿Ô´Ù ³ª°£°Å Ã¼Å© ==========================
// 
// º¯°æ : AUTO LOAD ÀÌ¹Ç·Î,  LOAD OK ¹Þ°í ALIGN ¿Ï·á·Î ¼öÁ¤
; L113
LOAD      M00201	// LF_AUTO RUN
AND       T2001	// IN-BUFF RIGT(L-LD)
AND NOT   P00014	// FRONT SAFETY SENSOR
OR        M18200	// ¿ÞÂÊ ¼Õµé¾î¿È
AND NOT   K00252	// LOADING ±â ONLINE
AND NOT   M18100	// L_IN BUFFER VC ON
OUT       M18200	// ¿ÞÂÊ ¼Õµé¾î¿È
TON       T1190 200	// ¿ÞÂÊ ¼Õµé¾î¿È
; L115
LOAD      M00211	// RT_AUTO RUN
AND       T2000	// IN-BUFF LEFT(R-LD)
AND NOT   P00014	// FRONT SAFETY SENSOR
OR        M18201	// ¿À¸¥ÂÊ ¼Õµé¾î¿È
AND NOT   K00252	// LOADING ±â ONLINE
AND NOT   M18600	// R_IN BUFFER VC ON
OUT       M18201	// ¿À¸¥ÂÊ ¼Õµé¾î¿È
TON       T1191 200	// ¿À¸¥ÂÊ ¼Õµé¾î¿È
// output comment: ¼öµ¿ÅõÀÔÇüÅÂ Àåºñ¿¡ ÅõÀÔºÎ ºö¼¾¼­°¡ 1°³·Î º¯°æ(2021.12)
; L117
LOAD      P00014	// FRONT SAFETY SENSOR
AND       T1190	// ¿ÞÂÊ ¼Õµé¾î¿È
AND       T2001	// IN-BUFF RIGT(L-LD)
AND       P0002D	// L_IN BUFF ROTATE-LD
AND NOT   K00252	// LOADING ±â ONLINE
OUT       M18202	// ¿ÞÂÊ ¼Õ³ª°¨
// output comment: ±âÁ¸ ÀÛ¾÷ÀÚ ¼Õ ºüÁ® ³ª°¡´Â°Í °¨ÁöÇØ¼­ Áø°ø ÇÏ´ø°ÍÀ» AUTO LOAD ÈÄ ALIGN µ¿ÀÛ ÇÏ¸é Áø°øÇÏ°Ô ¼öÁ¤
; L118
LOAD      P00014	// FRONT SAFETY SENSOR
AND       T1191	// ¿À¸¥ÂÊ ¼Õµé¾î¿È
AND       T2000	// IN-BUFF LEFT(R-LD)
AND       P0006D	// R_IN BUFF ROTATE-LD
AND NOT   K00252	// LOADING ±â ONLINE
OUT       M18204	// ¿À¸¥ÂÊ ¼Õ³ª°¨
// output comment: ¼öµ¿ÅõÀÔÇüÅÂ Àåºñ¿¡ ÅõÀÔºÎ ºö¼¾¼­°¡ 1°³·Î º¯°æ(2021.12)
// ======================== ENABLE ==========================
; L120
LOAD      M06510	// L_IN BUFFER DIE VACUUM CHECK ON
OR        M00082	// ÀÚÀç¹èÃâ IN_BUFFER ÅõÀÔ 
OR        M1902F	// DRY RUN
OUT       M1817A	// L_IN BUFFER DIE VACUUM CHECK ON

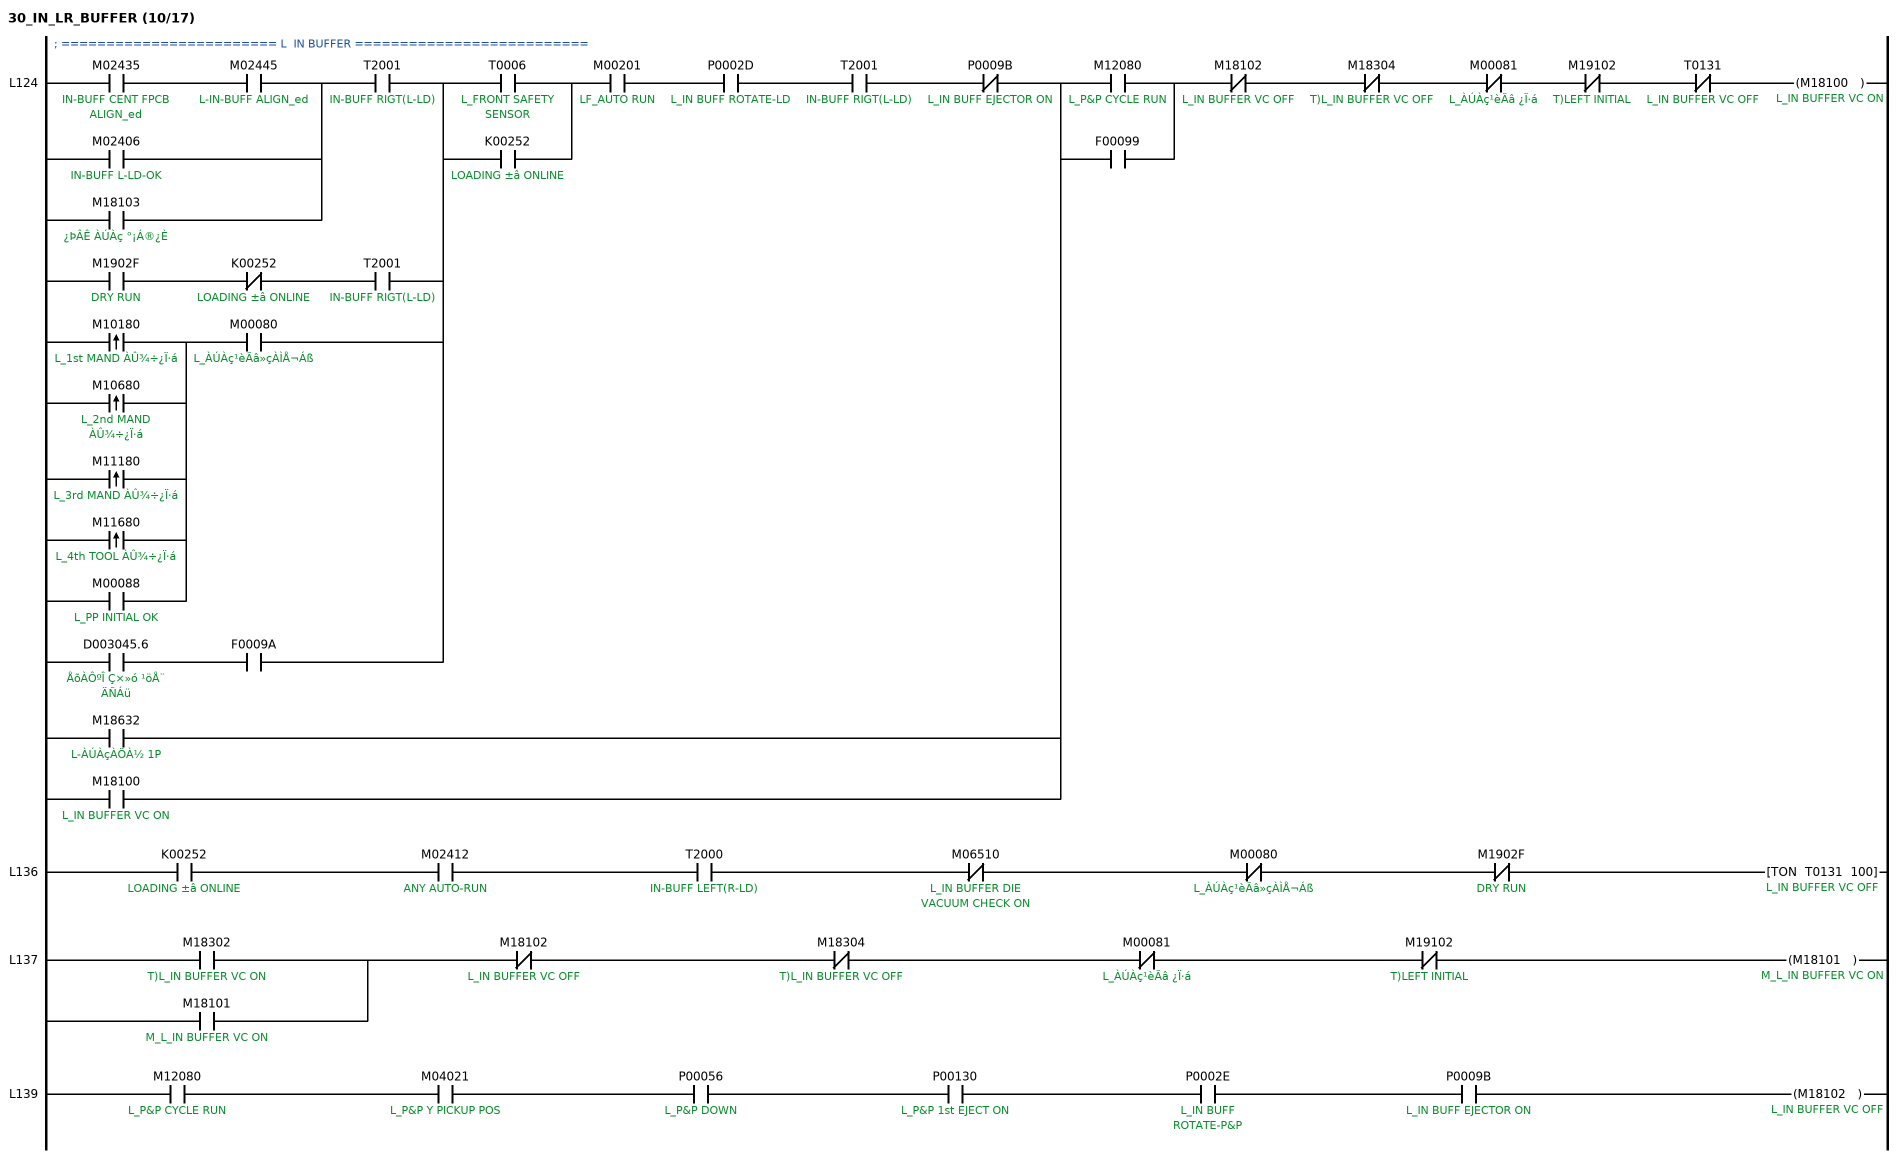
// ======================== L  IN BUFFER ==========================
; L124
LOAD      M02435	// IN-BUFF CENT FPCB ALIGN_ed
AND       M02445	// L-IN-BUFF ALIGN_ed
OR        M02406	// IN-BUFF L-LD-OK
OR        M18103	// ¿ÞÂÊ ÀÚÀç °¡Á®¿È
AND       T2001	// IN-BUFF RIGT(L-LD)
LOAD      M1902F	// DRY RUN
AND NOT   K00252	// LOADING ±â ONLINE
AND       T2001	// IN-BUFF RIGT(L-LD)
OR LOAD
LOADP     M10180	// L_1st MAND ÀÛ¾÷¿Ï·á
ORP       M10680	// L_2nd MAND ÀÛ¾÷¿Ï·á
ORP       M11180	// L_3rd MAND ÀÛ¾÷¿Ï·á
ORP       M11680	// L_4th TOOL ÀÛ¾÷¿Ï·á
OR        M00088	// L_PP INITIAL OK
AND       M00080	// L_ÀÚÀç¹èÃâ»çÀÌÅ¬Áß
OR LOAD
LOAD      D003045.6	// ÅõÀÔºÎ Ç×»ó ¹öÅ¨ ÄÑÁü
AND       F0009A
OR LOAD
LOAD      T0006	// L_FRONT SAFETY SENSOR
OR        K00252	// LOADING ±â ONLINE
AND LOAD
AND       M00201	// LF_AUTO RUN
AND       P0002D	// L_IN BUFF ROTATE-LD
AND       T2001	// IN-BUFF RIGT(L-LD)
AND NOT   P0009B	// L_IN BUFF EJECTOR ON
OR        M18632	// L-ÀÚÀçÀÖÀ½ 1P
OR        M18100	// L_IN BUFFER VC ON
LOAD      M12080	// L_P&P CYCLE RUN
OR        F00099
AND LOAD
AND NOT   M18102	// L_IN BUFFER VC OFF
AND NOT   M18304	// T)L_IN BUFFER VC OFF
AND NOT   M00081	// L_ÀÚÀç¹èÃâ ¿Ï·á
AND NOT   M19102	// T)LEFT INITIAL
AND NOT   T0131	// L_IN BUFFER VC OFF
OUT       M18100	// L_IN BUFFER VC ON
; L136
LOAD      K00252	// LOADING ±â ONLINE
AND       M02412	// ANY AUTO-RUN
AND       T2000	// IN-BUFF LEFT(R-LD)
AND NOT   M06510	// L_IN BUFFER DIE VACUUM CHECK ON
AND NOT   M00080	// L_ÀÚÀç¹èÃâ»çÀÌÅ¬Áß
AND NOT   M1902F	// DRY RUN
TON       T0131 100	// L_IN BUFFER VC OFF
; L137
LOAD      M18302	// T)L_IN BUFFER VC ON
OR        M18101	// M_L_IN BUFFER VC ON
AND NOT   M18102	// L_IN BUFFER VC OFF
AND NOT   M18304	// T)L_IN BUFFER VC OFF
AND NOT   M00081	// L_ÀÚÀç¹èÃâ ¿Ï·á
AND NOT   M19102	// T)LEFT INITIAL
OUT       M18101	// M_L_IN BUFFER VC ON
; L139
LOAD      M12080	// L_P&P CYCLE RUN
AND       M04021	// L_P&P Y PICKUP POS
AND       P00056	// L_P&P DOWN
AND       P00130	// L_P&P 1st EJECT ON
AND       P0002E	// L_IN BUFF ROTATE-P&P
AND       P0009B	// L_IN BUFF EJECTOR ON
OUT       M18102	// L_IN BUFFER VC OFF

